LIN {X -0.060,Y -618.449,Z 1038.668,A 0.000,B 0.000,C 90.000,E1 336.230} C_DIS
LIN {X 0.200,Y -620.770,Z 1038.662,A 0.000,B 0.000,C 90.000,E1 335.177} C_DIS
LIN {X 0.196,Y -624.173,Z 1038.652,A 0.000,B 0.000,C 90.000,E1 333.384} C_DIS
LIN {X 0.244,Y -626.247,Z 1038.645,A 0.000,B 0.000,C 90.000,E1 332.103} C_DIS
LIN {X -0.253,Y -627.737,Z 1038.640,A 0.000,B 0.000,C 90.000,E1 331.129} C_DIS
LIN {X -0.406,Y -629.343,Z 1038.632,A 0.000,B 0.000,C 90.000,E1 329.871} C_DIS
LIN {X 0.333,Y -630.595,Z 1038.625,A 0.000,B 0.000,C 90.000,E1 328.535} C_DIS
LIN {X 0.027,Y -631.655,Z 1038.618,A 0.000,B 0.000,C 90.000,E1 327.296} C_DIS
LIN {X 0.271,Y -632.422,Z 1038.611,A 0.000,B 0.000,C 90.000,E1 326.008} C_DIS
LIN {X -0.015,Y -632.715,Z 1038.606,A 0.000,B 0.000,C 90.000,E1 325.022} C_DIS
LIN {X 0.076,Y -632.913,Z 1038.597,A 0.000,B 0.000,C 90.000,E1 323.497} C_DIS
LIN {X -0.098,Y -633.067,Z 1038.587,A 0.000,B 0.000,C 90.000,E1 321.743} C_DIS
LIN {X 0.257,Y -633.344,Z 1038.579,A 0.000,B 0.000,C 90.000,E1 320.194} C_DIS
LIN {X 0.129,Y -633.583,Z 1038.571,A 0.000,B 0.000,C 90.000,E1 318.690} C_DIS
LIN {X -0.259,Y -633.721,Z 1038.565,A 0.000,B 0.000,C 90.000,E1 317.715} C_DIS
LIN {X 0.356,Y -634.009,Z 1038.555,A 0.000,B 0.000,C 90.000,E1 315.891} C_DIS
LIN {X -0.368,Y -634.348,Z 1038.545,A 0.000,B 0.000,C 90.000,E1 314.190} C_DIS
LIN {X 0.114,Y -634.612,Z 1038.540,A 0.000,B 0.000,C 90.000,E1 313.137} C_DIS
LIN {X -0.371,Y -634.828,Z 1038.533,A 0.000,B 0.000,C 90.000,E1 311.919} C_DIS
LIN {X 0.051,Y -634.991,Z 1038.526,A 0.000,B 0.000,C 90.000,E1 310.620} C_DIS
LIN {X 0.204,Y -635.096,Z 1038.521,A 0.000,B 0.000,C 90.000,E1 309.850} C_DIS
LIN {X 0.329,Y -635.110,Z 1038.516,A 0.000,B 0.000,C 90.000,E1 308.830} C_DIS
LIN {X 0.074,Y -635.210,Z 1038.503,A 0.000,B 0.000,C 90.000,E1 306.583} C_DIS
LIN {X -0.174,Y -635.840,Z 1038.488,A 0.000,B 0.000,C 90.000,E1 303.833} C_DIS
LIN {X 0.041,Y -636.792,Z 1038.477,A 0.000,B 0.000,C 90.000,E1 301.799} C_DIS
LIN {X 0.088,Y -637.787,Z 1038.468,A 0.000,B 0.000,C 90.000,E1 300.285} C_DIS
LIN {X -0.030,Y -639.112,Z 1038.459,A 0.000,B 0.000,C 90.000,E1 298.537} C_DIS
LIN {X 0.261,Y -640.188,Z 1038.452,A 0.000,B 0.000,C 90.000,E1 297.257} C_DIS
LIN {X -0.061,Y -640.906,Z 1038.446,A 0.000,B 0.000,C 90.000,E1 296.283} C_DIS
LIN {X -0.147,Y -641.266,Z 1038.442,A 0.000,B 0.000,C 90.000,E1 295.540} C_DIS
LIN {X 0.117,Y -641.463,Z 1038.436,A 0.000,B 0.000,C 90.000,E1 294.515} C_DIS
LIN {X 0.111,Y -641.357,Z 1038.431,A 0.000,B 0.000,C 90.000,E1 293.515} C_DIS
LIN {X 0.102,Y -640.897,Z 1038.425,A 0.000,B 0.000,C 90.000,E1 292.514} C_DIS
LIN {X 0.029,Y -640.393,Z 1038.421,A 0.000,B 0.000,C 90.000,E1 291.770} C_DIS
LIN {X -0.154,Y -640.110,Z 1038.420,A 0.000,B 0.000,C 90.000,E1 291.535} C_DIS
LIN {X -0.284,Y -639.216,Z 1038.417,A 0.000,B 0.000,C 90.000,E1 291.046} C_DIS
LIN {X -0.192,Y -637.595,Z 1038.414,A 0.000,B 0.000,C 90.000,E1 290.536} C_DIS
LIN {X 0.222,Y -636.440,Z 1038.413,A 0.000,B 0.000,C 90.000,E1 290.248} C_DIS
LIN {X 0.069,Y -632.866,Z 1038.410,A 0.000,B 0.000,C 90.000,E1 289.758} C_DIS
LIN {X 0.078,Y -631.575,Z 1038.409,A 0.000,B 0.000,C 90.000,E1 289.631} C_DIS
LIN {X 0.157,Y -627.206,Z 1038.407,A 0.000,B 0.000,C 90.000,E1 289.268} C_DIS
LIN {X 0.365,Y -625.795,Z 1038.407,A 0.000,B 0.000,C 90.000,E1 289.141} C_DIS
LIN {X -0.222,Y -623.815,Z 1038.406,A 0.000,B 0.000,C 90.000,E1 289.087} C_DIS
LIN {X -0.131,Y -619.940,Z 1038.405,A 0.000,B 0.000,C 90.000,E1 288.906} C_DIS
LIN {X -0.205,Y -616.809,Z 1038.404,A 0.000,B 0.000,C 90.000,E1 288.725} C_DIS
LIN {X -0.172,Y -609.298,Z 1038.402,A 0.000,B 0.000,C 90.000,E1 288.417} C_DIS
LIN {X -0.167,Y -595.438,Z 1038.400,A 0.000,B 0.000,C 90.000,E1 287.928} C_DIS
LIN {X -0.153,Y -588.161,Z 1038.398,A 0.000,B 0.000,C 90.000,E1 287.692} C_DIS
LIN {X -0.073,Y -579.446,Z 1038.397,A 0.000,B 0.000,C 90.000,E1 287.402} C_DIS
LIN {X 0.070,Y -570.332,Z 1038.395,A 0.000,B 0.000,C 90.000,E1 287.040} C_DIS
LIN {X 0.055,Y -565.220,Z 1038.393,A 0.000,B 0.000,C 90.000,E1 286.804} C_DIS
LIN {X -0.217,Y -562.660,Z 1038.393,A 0.000,B 0.000,C 90.000,E1 286.677} C_DIS
LIN {X 0.099,Y -559.516,Z 1038.391,A 0.000,B 0.000,C 90.000,E1 286.441} C_DIS
LIN {X 0.192,Y -558.622,Z 1038.391,A 0.000,B 0.000,C 90.000,E1 286.315} C_DIS
LIN {X -0.205,Y -558.386,Z 1038.391,A 0.000,B 0.000,C 90.000,E1 286.315} C_DIS
LIN {X 0.290,Y -586.431,Z 1038.391,A 0.000,B 0.000,C 90.000,E1 286.260} C_DIS
LIN {X -0.354,Y -591.713,Z 1038.390,A 0.000,B 0.000,C 90.000,E1 286.205} C_DIS
LIN {X 0.109,Y -594.085,Z 1038.389,A 0.000,B 0.000,C 90.000,E1 286.079} C_DIS
LIN {X 0.215,Y -598.623,Z 1038.388,A 0.000,B 0.000,C 90.000,E1 285.733} C_DIS
LIN {X -0.132,Y -600.931,Z 1038.386,A 0.000,B 0.000,C 90.000,E1 285.552} C_DIS
LIN {X -0.291,Y -604.296,Z 1038.384,A 0.000,B 0.000,C 90.000,E1 285.190} C_DIS
LIN {X 0.020,Y -606.088,Z 1038.383,A 0.000,B 0.000,C 90.000,E1 284.898} C_DIS
LIN {X 0.233,Y -609.291,Z 1038.380,A 0.000,B 0.000,C 90.000,E1 284.356} C_DIS
LIN {X 0.115,Y -612.175,Z 1038.376,A 0.000,B 0.000,C 90.000,E1 283.716} C_DIS
LIN {X 0.359,Y -614.055,Z 1038.373,A 0.000,B 0.000,C 90.000,E1 283.175} C_DIS
LIN {X 0.115,Y -614.648,Z 1038.372,A 0.000,B 0.000,C 90.000,E1 282.939} C_DIS
LIN {X 0.233,Y -615.426,Z 1038.369,A 0.000,B 0.000,C 90.000,E1 282.411} C_DIS
LIN {X 0.230,Y -615.605,Z 1038.366,A 0.000,B 0.000,C 90.000,E1 281.895} C_DIS
LIN {X -0.244,Y -615.085,Z 1038.363,A 0.000,B 0.000,C 90.000,E1 281.422} C_DIS
LIN {X 0.121,Y -614.650,Z 1038.362,A 0.000,B 0.000,C 90.000,E1 281.130} C_DIS
LIN {X 0.242,Y -613.270,Z 1038.359,A 0.000,B 0.000,C 90.000,E1 280.602} C_DIS
LIN {X 0.240,Y -610.812,Z 1038.356,A 0.000,B 0.000,C 90.000,E1 280.084} C_DIS
LIN {X -0.269,Y -607.576,Z 1038.353,A 0.000,B 0.000,C 90.000,E1 279.613} C_DIS
LIN {X 0.065,Y -605.581,Z 1038.352,A 0.000,B 0.000,C 90.000,E1 279.321} C_DIS
LIN {X -0.142,Y -603.544,Z 1038.350,A 0.000,B 0.000,C 90.000,E1 279.095} C_DIS
LIN {X -0.232,Y -602.339,Z 1038.350,A 0.000,B 0.000,C 90.000,E1 278.973} C_DIS
LIN {X 0.150,Y -599.442,Z 1038.348,A 0.000,B 0.000,C 90.000,E1 278.690} C_DIS
LIN {X 0.085,Y -597.004,Z 1038.347,A 0.000,B 0.000,C 90.000,E1 278.454} C_DIS
LIN {X 0.092,Y -592.425,Z 1038.345,A 0.000,B 0.000,C 90.000,E1 278.106} C_DIS
LIN {X -0.161,Y -590.174,Z 1038.344,A 0.000,B 0.000,C 90.000,E1 277.936} C_DIS
LIN {X -0.137,Y -588.118,Z 1038.343,A 0.000,B 0.000,C 90.000,E1 277.814} C_DIS
LIN {X -0.193,Y -585.716,Z 1038.343,A 0.000,B 0.000,C 90.000,E1 277.701} C_DIS
LIN {X -0.111,Y -582.851,Z 1038.342,A 0.000,B 0.000,C 90.000,E1 277.530} C_DIS
LIN {X 0.253,Y -580.858,Z 1038.341,A 0.000,B 0.000,C 90.000,E1 277.409} C_DIS
LIN {X -0.022,Y -576.101,Z 1038.341,A 0.000,B 0.000,C 90.000,E1 277.296} C_DIS
LIN {X 0.270,Y -574.938,Z 1038.340,A 0.000,B 0.000,C 90.000,E1 277.239} C_DIS
LIN {X -0.235,Y -568.564,Z 1038.340,A 0.000,B 0.000,C 90.000,E1 277.239} C_DIS
LIN {X -0.270,Y -546.914,Z 1038.340,A 0.000,B 0.000,C 90.000,E1 277.239} C_DIS
LIN {X -0.073,Y -545.872,Z 1038.339,A 0.000,B 0.000,C 90.000,E1 277.068} C_DIS
LIN {X 0.058,Y -543.522,Z 1038.338,A 0.000,B 0.000,C 90.000,E1 276.777} C_DIS
LIN {X 0.016,Y -543.511,Z 1038.338,A 0.000,B 0.000,C 90.000,E1 276.777} C_DIS
LIN {X -0.061,Y -542.122,Z 1038.331,A 0.000,B 0.000,C 90.000,E1 275.511} C_DIS
LIN {X 0.194,Y -540.725,Z 1038.320,A 0.000,B 0.000,C 90.000,E1 273.498} C_DIS
LIN {X -0.170,Y -539.690,Z 1038.309,A 0.000,B 0.000,C 90.000,E1 271.547} C_DIS
LIN {X -0.101,Y -539.052,Z 1038.302,A 0.000,B 0.000,C 90.000,E1 270.401} C_DIS
LIN {X -0.026,Y -538.094,Z 1038.294,A 0.000,B 0.000,C 90.000,E1 268.969} C_DIS
LIN {X 0.054,Y -536.613,Z 1038.283,A 0.000,B 0.000,C 90.000,E1 266.963} C_DIS
LIN {X 0.125,Y -535.600,Z 1038.275,A 0.000,B 0.000,C 90.000,E1 265.527} C_DIS
LIN {X 0.220,Y -534.366,Z 1038.266,A 0.000,B 0.000,C 90.000,E1 263.799} C_DIS
LIN {X -0.264,Y -533.403,Z 1038.259,A 0.000,B 0.000,C 90.000,E1 262.704} C_DIS
LIN {X -0.121,Y -531.960,Z 1038.251,A 0.000,B 0.000,C 90.000,E1 261.254} C_DIS
LIN {X 0.109,Y -529.384,Z 1038.239,A 0.000,B 0.000,C 90.000,E1 258.926} C_DIS
LIN {X -0.212,Y -527.530,Z 1038.229,A 0.000,B 0.000,C 90.000,E1 257.229} C_DIS
LIN {X 0.050,Y -525.635,Z 1038.219,A 0.000,B 0.000,C 90.000,E1 255.463} C_DIS
LIN {X -0.116,Y -524.030,Z 1038.211,A 0.000,B 0.000,C 90.000,E1 254.031} C_DIS
LIN {X 0.192,Y -522.504,Z 1038.203,A 0.000,B 0.000,C 90.000,E1 252.543} C_DIS
LIN {X -0.026,Y -521.203,Z 1038.197,A 0.000,B 0.000,C 90.000,E1 251.402} C_DIS
LIN {X 0.018,Y -519.076,Z 1038.187,A 0.000,B 0.000,C 90.000,E1 249.645} C_DIS
LIN {X -0.096,Y -516.889,Z 1038.177,A 0.000,B 0.000,C 90.000,E1 247.901} C_DIS
LIN {X -0.232,Y -515.322,Z 1038.171,A 0.000,B 0.000,C 90.000,E1 246.741} C_DIS
LIN {X -0.113,Y -514.169,Z 1038.166,A 0.000,B 0.000,C 90.000,E1 245.845} C_DIS
LIN {X 0.015,Y -511.805,Z 1038.158,A 0.000,B 0.000,C 90.000,E1 244.357} C_DIS
LIN {X -0.025,Y -509.920,Z 1038.151,A 0.000,B 0.000,C 90.000,E1 243.179} C_DIS
LIN {X 0.133,Y -507.929,Z 1038.144,A 0.000,B 0.000,C 90.000,E1 241.975} C_DIS
LIN {X -0.077,Y -505.267,Z 1038.136,A 0.000,B 0.000,C 90.000,E1 240.511} C_DIS
LIN {X 0.110,Y -502.587,Z 1038.128,A 0.000,B 0.000,C 90.000,E1 238.997} C_DIS
LIN {X 0.096,Y -499.218,Z 1038.118,A 0.000,B 0.000,C 90.000,E1 237.199} C_DIS
LIN {X -0.015,Y -496.865,Z 1038.111,A 0.000,B 0.000,C 90.000,E1 236.008} C_DIS
LIN {X -0.034,Y -492.964,Z 1038.101,A 0.000,B 0.000,C 90.000,E1 234.196} C_DIS
LIN {X -0.092,Y -489.440,Z 1038.093,A 0.000,B 0.000,C 90.000,E1 232.683} C_DIS
LIN {X -0.056,Y -483.684,Z 1038.079,A 0.000,B 0.000,C 90.000,E1 230.231} C_DIS
LIN {X -0.125,Y -478.929,Z 1038.067,A 0.000,B 0.000,C 90.000,E1 228.081} C_DIS
LIN {X -0.202,Y -475.740,Z 1038.058,A 0.000,B 0.000,C 90.000,E1 226.539} C_DIS
LIN {X -0.166,Y -471.201,Z 1038.046,A 0.000,B 0.000,C 90.000,E1 224.352} C_DIS
LIN {X 0.081,Y -466.692,Z 1038.034,A 0.000,B 0.000,C 90.000,E1 222.123} C_DIS
LIN {X 0.122,Y -463.522,Z 1038.025,A 0.000,B 0.000,C 90.000,E1 220.539} C_DIS
LIN {X -0.158,Y -459.461,Z 1038.015,A 0.000,B 0.000,C 90.000,E1 218.669} C_DIS
LIN {X -0.187,Y -455.999,Z 1038.006,A 0.000,B 0.000,C 90.000,E1 217.076} C_DIS
LIN {X 0.077,Y -452.503,Z 1037.997,A 0.000,B 0.000,C 90.000,E1 215.438} C_DIS
LIN {X -0.035,Y -450.542,Z 1037.992,A 0.000,B 0.000,C 90.000,E1 214.485} C_DIS
LIN {X -0.066,Y -446.481,Z 1037.981,A 0.000,B 0.000,C 90.000,E1 212.546} C_DIS
LIN {X -0.065,Y -442.186,Z 1037.970,A 0.000,B 0.000,C 90.000,E1 210.590} C_DIS
LIN {X -0.089,Y -439.234,Z 1037.963,A 0.000,B 0.000,C 90.000,E1 209.283} C_DIS
LIN {X -0.155,Y -436.188,Z 1037.955,A 0.000,B 0.000,C 90.000,E1 207.975} C_DIS
LIN {X -0.063,Y -431.773,Z 1037.944,A 0.000,B 0.000,C 90.000,E1 205.976} C_DIS
LIN {X 0.113,Y -426.007,Z 1037.929,A 0.000,B 0.000,C 90.000,E1 203.281} C_DIS
LIN {X -0.057,Y -420.811,Z 1037.915,A 0.000,B 0.000,C 90.000,E1 200.610} C_DIS
LIN {X -0.196,Y -413.886,Z 1037.890,A 0.000,B 0.000,C 90.000,E1 196.205} C_DIS
LIN {X -0.121,Y -411.969,Z 1037.880,A 0.000,B 0.000,C 90.000,E1 194.481} C_DIS
LIN {X 0.161,Y -411.252,Z 1037.875,A 0.000,B 0.000,C 90.000,E1 193.411} C_DIS
LIN {X -0.066,Y -410.760,Z 1037.869,A 0.000,B 0.000,C 90.000,E1 192.411} C_DIS
LIN {X -0.010,Y -411.012,Z 1037.865,A 0.000,B 0.000,C 90.000,E1 191.715} C_DIS
LIN {X 0.020,Y -411.285,Z 1037.863,A 0.000,B 0.000,C 90.000,E1 191.366} C_DIS
LIN {X 0.130,Y -411.738,Z 1037.861,A 0.000,B 0.000,C 90.000,E1 191.007} C_DIS
LIN {X -0.141,Y -413.356,Z 1037.858,A 0.000,B 0.000,C 90.000,E1 190.366} C_DIS
LIN {X -0.105,Y -414.633,Z 1037.856,A 0.000,B 0.000,C 90.000,E1 190.018} C_DIS
LIN {X -0.071,Y -416.767,Z 1037.853,A 0.000,B 0.000,C 90.000,E1 189.500} C_DIS
LIN {X -0.076,Y -419.086,Z 1037.850,A 0.000,B 0.000,C 90.000,E1 189.095} C_DIS
LIN {X 0.050,Y -422.248,Z 1037.848,A 0.000,B 0.000,C 90.000,E1 188.568} C_DIS
LIN {X -0.094,Y -435.430,Z 1037.838,A 0.000,B 0.000,C 90.000,E1 186.777} C_DIS
LIN {X -0.176,Y -442.951,Z 1037.832,A 0.000,B 0.000,C 90.000,E1 185.796} C_DIS
LIN {X 0.050,Y -453.968,Z 1037.824,A 0.000,B 0.000,C 90.000,E1 184.302} C_DIS
LIN {X -0.211,Y -462.264,Z 1037.818,A 0.000,B 0.000,C 90.000,E1 183.212} C_DIS
LIN {X -0.110,Y -472.302,Z 1037.810,A 0.000,B 0.000,C 90.000,E1 181.776} C_DIS
LIN {X 0.235,Y -481.700,Z 1037.802,A 0.000,B 0.000,C 90.000,E1 180.344} C_DIS
LIN {X 0.172,Y -487.705,Z 1037.797,A 0.000,B 0.000,C 90.000,E1 179.427} C_DIS
LIN {X -0.149,Y -494.571,Z 1037.791,A 0.000,B 0.000,C 90.000,E1 178.396} C_DIS
LIN {X -0.056,Y -500.306,Z 1037.786,A 0.000,B 0.000,C 90.000,E1 177.478} C_DIS
LIN {X 0.111,Y -507.412,Z 1037.779,A 0.000,B 0.000,C 90.000,E1 176.274} C_DIS
LIN {X 0.222,Y -516.017,Z 1037.771,A 0.000,B 0.000,C 90.000,E1 174.780} C_DIS
LIN {X 0.026,Y -524.489,Z 1037.763,A 0.000,B 0.000,C 90.000,E1 173.337} C_DIS
LIN {X -0.017,Y -532.743,Z 1037.755,A 0.000,B 0.000,C 90.000,E1 171.894} C_DIS
LIN {X -0.112,Y -541.531,Z 1037.746,A 0.000,B 0.000,C 90.000,E1 170.330} C_DIS
LIN {X 0.057,Y -550.142,Z 1037.738,A 0.000,B 0.000,C 90.000,E1 168.757} C_DIS
LIN {X -0.007,Y -558.485,Z 1037.729,A 0.000,B 0.000,C 90.000,E1 167.229} C_DIS
LIN {X 0.299,Y -563.558,Z 1037.724,A 0.000,B 0.000,C 90.000,E1 166.228} C_DIS
LIN {X 0.181,Y -570.648,Z 1037.716,A 0.000,B 0.000,C 90.000,E1 164.866} C_DIS
LIN {X 0.081,Y -575.369,Z 1037.711,A 0.000,B 0.000,C 90.000,E1 163.921} C_DIS
LIN {X 0.198,Y -579.985,Z 1037.705,A 0.000,B 0.000,C 90.000,E1 162.960} C_DIS
LIN {X -0.184,Y -584.304,Z 1037.700,A 0.000,B 0.000,C 90.000,E1 162.054} C_DIS
LIN {X -0.032,Y -588.964,Z 1037.694,A 0.000,B 0.000,C 90.000,E1 160.967} C_DIS
LIN {X 0.066,Y -594.393,Z 1037.687,A 0.000,B 0.000,C 90.000,E1 159.625} C_DIS
LIN {X -0.211,Y -598.419,Z 1037.681,A 0.000,B 0.000,C 90.000,E1 158.592} C_DIS
LIN {X 0.262,Y -603.058,Z 1037.674,A 0.000,B 0.000,C 90.000,E1 157.230} C_DIS
LIN {X -0.238,Y -606.530,Z 1037.668,A 0.000,B 0.000,C 90.000,E1 156.230} C_DIS
LIN {X -0.143,Y -609.792,Z 1037.662,A 0.000,B 0.000,C 90.000,E1 155.177} C_DIS
LIN {X -0.305,Y -612.814,Z 1037.656,A 0.000,B 0.000,C 90.000,E1 154.152} C_DIS
LIN {X 0.104,Y -616.332,Z 1037.649,A 0.000,B 0.000,C 90.000,E1 152.820} C_DIS
LIN {X 0.319,Y -619.009,Z 1037.643,A 0.000,B 0.000,C 90.000,E1 151.769} C_DIS
LIN {X 0.031,Y -622.879,Z 1037.635,A 0.000,B 0.000,C 90.000,E1 150.255} C_DIS
LIN {X -0.190,Y -626.033,Z 1037.628,A 0.000,B 0.000,C 90.000,E1 148.997} C_DIS
LIN {X -0.034,Y -629.093,Z 1037.621,A 0.000,B 0.000,C 90.000,E1 147.709} C_DIS
LIN {X 0.185,Y -632.629,Z 1037.612,A 0.000,B 0.000,C 90.000,E1 146.167} C_DIS
LIN {X -0.231,Y -636.111,Z 1037.604,A 0.000,B 0.000,C 90.000,E1 144.689} C_DIS
LIN {X 0.317,Y -639.575,Z 1037.595,A 0.000,B 0.000,C 90.000,E1 143.130} C_DIS
LIN {X -0.081,Y -643.088,Z 1037.587,A 0.000,B 0.000,C 90.000,E1 141.662} C_DIS
LIN {X 0.010,Y -647.078,Z 1037.577,A 0.000,B 0.000,C 90.000,E1 139.908} C_DIS
LIN {X 0.108,Y -651.094,Z 1037.568,A 0.000,B 0.000,C 90.000,E1 138.162} C_DIS
LIN {X -0.268,Y -656.433,Z 1037.555,A 0.000,B 0.000,C 90.000,E1 135.972} C_DIS
LIN {X -0.054,Y -663.721,Z 1037.540,A 0.000,B 0.000,C 90.000,E1 133.257} C_DIS
LIN {X -0.098,Y -667.183,Z 1037.534,A 0.000,B 0.000,C 90.000,E1 132.043} C_DIS
LIN {X -0.048,Y -670.668,Z 1037.527,A 0.000,B 0.000,C 90.000,E1 130.825} C_DIS
LIN {X 0.156,Y -674.730,Z 1037.519,A 0.000,B 0.000,C 90.000,E1 129.358} C_DIS
LIN {X -0.097,Y -678.022,Z 1037.512,A 0.000,B 0.000,C 90.000,E1 128.177} C_DIS
LIN {X -0.139,Y -682.350,Z 1037.503,A 0.000,B 0.000,C 90.000,E1 126.503} C_DIS
LIN {X 0.432,Y -686.073,Z 1037.495,A 0.000,B 0.000,C 90.000,E1 125.025} C_DIS
LIN {X 0.116,Y -689.677,Z 1037.487,A 0.000,B 0.000,C 90.000,E1 123.627} C_DIS
LIN {X 0.065,Y -693.179,Z 1037.479,A 0.000,B 0.000,C 90.000,E1 122.212} C_DIS
LIN {X 0.192,Y -695.373,Z 1037.474,A 0.000,B 0.000,C 90.000,E1 121.258} C_DIS
LIN {X 0.241,Y -697.851,Z 1037.467,A 0.000,B 0.000,C 90.000,E1 120.079} C_DIS
LIN {X -0.193,Y -699.002,Z 1037.463,A 0.000,B 0.000,C 90.000,E1 119.411} C_DIS
LIN {X -0.085,Y -700.557,Z 1037.457,A 0.000,B 0.000,C 90.000,E1 118.231} C_DIS
LIN {X -0.350,Y -702.425,Z 1037.448,A 0.000,B 0.000,C 90.000,E1 116.616} C_DIS
LIN {X 0.116,Y -703.430,Z 1037.441,A 0.000,B 0.000,C 90.000,E1 115.412} C_DIS
LIN {X 0.031,Y -703.903,Z 1037.437,A 0.000,B 0.000,C 90.000,E1 114.719} C_DIS
LIN {X -0.044,Y -703.825,Z 1037.435,A 0.000,B 0.000,C 90.000,E1 114.259} C_DIS
LIN {X -0.049,Y -703.663,Z 1037.433,A 0.000,B 0.000,C 90.000,E1 114.027} C_DIS
LIN {X -0.131,Y -702.667,Z 1037.431,A 0.000,B 0.000,C 90.000,E1 113.567} C_DIS
LIN {X -0.134,Y -701.822,Z 1037.430,A 0.000,B 0.000,C 90.000,E1 113.334} C_DIS
LIN {X 0.138,Y -699.031,Z 1037.427,A 0.000,B 0.000,C 90.000,E1 112.845} C_DIS
LIN {X -0.374,Y -698.143,Z 1037.426,A 0.000,B 0.000,C 90.000,E1 112.770} C_DIS
LIN {X -0.242,Y -696.824,Z 1037.426,A 0.000,B 0.000,C 90.000,E1 112.642} C_DIS
LIN {X 0.161,Y -692.932,Z 1037.424,A 0.000,B 0.000,C 90.000,E1 112.386} C_DIS
LIN {X 0.326,Y -689.873,Z 1037.424,A 0.000,B 0.000,C 90.000,E1 112.206} C_DIS
LIN {X -0.046,Y -688.040,Z 1037.423,A 0.000,B 0.000,C 90.000,E1 112.153} C_DIS
LIN {X -0.156,Y -685.469,Z 1037.423,A 0.000,B 0.000,C 90.000,E1 112.078} C_DIS
LIN {X -0.191,Y -682.766,Z 1037.422,A 0.000,B 0.000,C 90.000,E1 112.025} C_DIS
LIN {X 0.323,Y -675.461,Z 1037.422,A 0.000,B 0.000,C 90.000,E1 111.897} C_DIS
LIN {X 0.249,Y -611.830,Z 1037.422,A 0.000,B 0.000,C 90.000,E1 111.897} C_DIS
LIN {X -0.103,Y -603.967,Z 1037.420,A 0.000,B 0.000,C 90.000,E1 111.663} C_DIS
LIN {X -0.084,Y -597.881,Z 1037.419,A 0.000,B 0.000,C 90.000,E1 111.354} C_DIS
LIN {X 0.117,Y -592.278,Z 1037.417,A 0.000,B 0.000,C 90.000,E1 110.972} C_DIS
LIN {X 0.178,Y -585.389,Z 1037.414,A 0.000,B 0.000,C 90.000,E1 110.429} C_DIS
LIN {X -0.147,Y -577.122,Z 1037.410,A 0.000,B 0.000,C 90.000,E1 109.758} C_DIS
LIN {X 0.193,Y -571.004,Z 1037.407,A 0.000,B 0.000,C 90.000,E1 109.268} C_DIS
LIN {X -0.352,Y -569.434,Z 1037.407,A 0.000,B 0.000,C 90.000,E1 109.214} C_DIS
LIN {X -0.255,Y -561.218,Z 1037.404,A 0.000,B 0.000,C 90.000,E1 108.725} C_DIS
LIN {X -0.158,Y -554.609,Z 1037.402,A 0.000,B 0.000,C 90.000,E1 108.362} C_DIS
LIN {X 0.138,Y -549.479,Z 1037.400,A 0.000,B 0.000,C 90.000,E1 108.000} C_DIS
LIN {X 0.108,Y -548.012,Z 1037.399,A 0.000,B 0.000,C 90.000,E1 107.819} C_DIS
LIN {X 0.067,Y -547.994,Z 1037.399,A 0.000,B 0.000,C 90.000,E1 107.819} C_DIS
LIN {X -0.157,Y -547.523,Z 1037.398,A 0.000,B 0.000,C 90.000,E1 107.583} C_DIS
LIN {X -0.026,Y -547.592,Z 1037.394,A 0.000,B 0.000,C 90.000,E1 106.985} C_DIS
LIN {X 0.031,Y -548.185,Z 1037.390,A 0.000,B 0.000,C 90.000,E1 106.134} C_DIS
LIN {X 0.044,Y -549.401,Z 1037.377,A 0.000,B 0.000,C 90.000,E1 103.883} C_DIS
LIN {X -0.230,Y -552.195,Z 1037.359,A 0.000,B 0.000,C 90.000,E1 100.546} C_DIS
LIN {X 0.138,Y -554.945,Z 1037.344,A 0.000,B 0.000,C 90.000,E1 97.992} C_DIS
LIN {X 0.068,Y -556.523,Z 1037.337,A 0.000,B 0.000,C 90.000,E1 96.606} C_DIS
LIN {X 0.020,Y -557.995,Z 1037.329,A 0.000,B 0.000,C 90.000,E1 95.220} C_DIS
LIN {X -0.182,Y -558.849,Z 1037.323,A 0.000,B 0.000,C 90.000,E1 94.131} C_DIS
LIN {X 0.107,Y -559.464,Z 1037.318,A 0.000,B 0.000,C 90.000,E1 93.269} C_DIS
LIN {X 0.131,Y -560.249,Z 1037.309,A 0.000,B 0.000,C 90.000,E1 91.604} C_DIS
LIN {X 0.134,Y -560.857,Z 1037.300,A 0.000,B 0.000,C 90.000,E1 89.943} C_DIS
LIN {X 0.264,Y -561.537,Z 1037.289,A 0.000,B 0.000,C 90.000,E1 87.993} C_DIS
LIN {X 0.213,Y -561.973,Z 1037.281,A 0.000,B 0.000,C 90.000,E1 86.617} C_DIS
LIN {X -0.261,Y -562.515,Z 1037.272,A 0.000,B 0.000,C 90.000,E1 85.008} C_DIS
LIN {X -0.265,Y -562.849,Z 1037.265,A 0.000,B 0.000,C 90.000,E1 83.628} C_DIS
LIN {X -0.218,Y -563.471,Z 1037.251,A 0.000,B 0.000,C 90.000,E1 81.141} C_DIS
LIN {X 0.041,Y -564.402,Z 1037.237,A 0.000,B 0.000,C 90.000,E1 78.634} C_DIS
LIN {X -0.112,Y -565.670,Z 1037.223,A 0.000,B 0.000,C 90.000,E1 76.172} C_DIS
LIN {X 0.251,Y -566.946,Z 1037.213,A 0.000,B 0.000,C 90.000,E1 74.212} C_DIS
LIN {X -0.067,Y -568.242,Z 1037.203,A 0.000,B 0.000,C 90.000,E1 72.598} C_DIS
LIN {X -0.150,Y -569.133,Z 1037.197,A 0.000,B 0.000,C 90.000,E1 71.511} C_DIS
LIN {X 0.127,Y -570.222,Z 1037.190,A 0.000,B 0.000,C 90.000,E1 70.115} C_DIS
LIN {X 0.062,Y -570.981,Z 1037.184,A 0.000,B 0.000,C 90.000,E1 69.028} C_DIS
LIN {X 0.031,Y -571.988,Z 1037.176,A 0.000,B 0.000,C 90.000,E1 67.667} C_DIS
LIN {X -0.150,Y -572.968,Z 1037.167,A 0.000,B 0.000,C 90.000,E1 66.049} C_DIS
LIN {X -0.239,Y -573.995,Z 1037.156,A 0.000,B 0.000,C 90.000,E1 64.152} C_DIS
LIN {X 0.259,Y -574.647,Z 1037.149,A 0.000,B 0.000,C 90.000,E1 62.743} C_DIS
LIN {X 0.254,Y -575.221,Z 1037.141,A 0.000,B 0.000,C 90.000,E1 61.385} C_DIS
LIN {X -0.275,Y -575.983,Z 1037.131,A 0.000,B 0.000,C 90.000,E1 59.537} C_DIS
LIN {X 0.176,Y -576.371,Z 1037.125,A 0.000,B 0.000,C 90.000,E1 58.408} C_DIS
LIN {X 0.287,Y -576.819,Z 1037.117,A 0.000,B 0.000,C 90.000,E1 57.041} C_DIS
LIN {X -0.070,Y -577.162,Z 1037.110,A 0.000,B 0.000,C 90.000,E1 55.722} C_DIS
LIN {X 0.068,Y -577.322,Z 1037.105,A 0.000,B 0.000,C 90.000,E1 54.895} C_DIS
LIN {X 0.054,Y -577.397,Z 1037.098,A 0.000,B 0.000,C 90.000,E1 53.543} C_DIS
LIN {X -0.277,Y -577.371,Z 1037.093,A 0.000,B 0.000,C 90.000,E1 52.763} C_DIS
LIN {X 0.039,Y -577.329,Z 1037.090,A 0.000,B 0.000,C 90.000,E1 52.190} C_DIS
LIN {X 0.058,Y -577.136,Z 1037.085,A 0.000,B 0.000,C 90.000,E1 51.376} C_DIS
LIN {X 0.093,Y -576.333,Z 1037.076,A 0.000,B 0.000,C 90.000,E1 49.747} C_DIS
LIN {X -0.188,Y -575.728,Z 1037.070,A 0.000,B 0.000,C 90.000,E1 48.690} C_DIS
LIN {X 0.192,Y -575.139,Z 1037.066,A 0.000,B 0.000,C 90.000,E1 47.838} C_DIS
LIN {X -0.010,Y -573.994,Z 1037.058,A 0.000,B 0.000,C 90.000,E1 46.500} C_DIS
LIN {X 0.348,Y -573.110,Z 1037.054,A 0.000,B 0.000,C 90.000,E1 45.648} C_DIS
LIN {X -0.306,Y -571.152,Z 1037.046,A 0.000,B 0.000,C 90.000,E1 44.352} C_DIS
LIN {X 0.110,Y -569.327,Z 1037.040,A 0.000,B 0.000,C 90.000,E1 43.218} C_DIS
LIN {X 0.105,Y -567.253,Z 1037.034,A 0.000,B 0.000,C 90.000,E1 42.123} C_DIS
LIN {X 0.009,Y -565.428,Z 1037.030,A 0.000,B 0.000,C 90.000,E1 41.310} C_DIS
LIN {X -0.056,Y -562.596,Z 1037.023,A 0.000,B 0.000,C 90.000,E1 40.216} C_DIS
LIN {X 0.141,Y -561.053,Z 1037.020,A 0.000,B 0.000,C 90.000,E1 39.644} C_DIS
LIN {X -0.009,Y -558.443,Z 1037.016,A 0.000,B 0.000,C 90.000,E1 38.830} C_DIS
LIN {X -0.187,Y -555.641,Z 1037.011,A 0.000,B 0.000,C 90.000,E1 38.016} C_DIS
LIN {X 0.042,Y -552.379,Z 1037.006,A 0.000,B 0.000,C 90.000,E1 37.156} C_DIS
LIN {X 0.234,Y -548.863,Z 1037.002,A 0.000,B 0.000,C 90.000,E1 36.297} C_DIS
LIN {X 0.066,Y -545.045,Z 1036.997,A 0.000,B 0.000,C 90.000,E1 35.471} C_DIS
LIN {X 0.169,Y -540.820,Z 1036.992,A 0.000,B 0.000,C 90.000,E1 34.612} C_DIS
LIN {X 0.061,Y -537.073,Z 1036.989,A 0.000,B 0.000,C 90.000,E1 33.913} C_DIS
LIN {X 0.068,Y -531.545,Z 1036.983,A 0.000,B 0.000,C 90.000,E1 32.911} C_DIS
LIN {X 0.031,Y -528.155,Z 1036.980,A 0.000,B 0.000,C 90.000,E1 32.339} C_DIS
LIN {X 0.250,Y -523.645,Z 1036.976,A 0.000,B 0.000,C 90.000,E1 31.592} C_DIS
LIN {X 0.155,Y -518.831,Z 1036.972,A 0.000,B 0.000,C 90.000,E1 30.875} C_DIS
LIN {X -0.251,Y -514.730,Z 1036.968,A 0.000,B 0.000,C 90.000,E1 30.335} C_DIS
LIN {X 0.279,Y -509.188,Z 1036.964,A 0.000,B 0.000,C 90.000,E1 29.539} C_DIS
LIN {X 0.245,Y -504.407,Z 1036.961,A 0.000,B 0.000,C 90.000,E1 28.949} C_DIS
LIN {X -0.144,Y -496.495,Z 1036.956,A 0.000,B 0.000,C 90.000,E1 28.103} C_DIS
LIN {X 0.172,Y -489.642,Z 1036.952,A 0.000,B 0.000,C 90.000,E1 27.334} C_DIS
LIN {X 0.131,Y -479.801,Z 1036.947,A 0.000,B 0.000,C 90.000,E1 26.360} C_DIS
LIN {X 0.173,Y -469.817,Z 1036.941,A 0.000,B 0.000,C 90.000,E1 25.412} C_DIS
LIN {X -0.155,Y -462.233,Z 1036.938,A 0.000,B 0.000,C 90.000,E1 24.771} C_DIS
LIN {X 0.239,Y -454.776,Z 1036.934,A 0.000,B 0.000,C 90.000,E1 24.079} C_DIS
LIN {X -0.148,Y -429.296,Z 1036.922,A 0.000,B 0.000,C 90.000,E1 21.897} C_DIS
LIN {X -0.083,Y -416.288,Z 1036.914,A 0.000,B 0.000,C 90.000,E1 20.610} C_DIS
LIN {X 0.084,Y -403.873,Z 1036.907,A 0.000,B 0.000,C 90.000,E1 19.214} C_DIS
LIN {X 0.163,Y -399.929,Z 1036.904,A 0.000,B 0.000,C 90.000,E1 18.725} C_DIS
LIN {X 0.068,Y -395.635,Z 1036.901,A 0.000,B 0.000,C 90.000,E1 18.127} C_DIS
LIN {X 0.024,Y -393.301,Z 1036.898,A 0.000,B 0.000,C 90.000,E1 17.692} C_DIS
LIN {X 0.128,Y -391.875,Z 1036.896,A 0.000,B 0.000,C 90.000,E1 17.166} C_DIS
LIN {X 0.139,Y -391.439,Z 1036.894,A 0.000,B 0.000,C 90.000,E1 16.804} C_DIS
LIN {X 0.163,Y -391.286,Z 1036.893,A 0.000,B 0.000,C 90.000,E1 16.622} C_DIS
LIN {X -0.152,Y -391.430,Z 1036.888,A 0.000,B 0.000,C 90.000,E1 15.898} C_DIS
LIN {X 0.189,Y -396.870,Z 1036.863,A 0.000,B 0.000,C 90.000,E1 11.243} C_DIS
LIN {X -0.056,Y -403.950,Z 1036.839,A 0.000,B 0.000,C 90.000,E1 7.068} C_DIS
LIN {X -0.113,Y -409.067,Z 1036.826,A 0.000,B 0.000,C 90.000,E1 4.645} C_DIS
LIN {X -0.144,Y -412.059,Z 1036.818,A 0.000,B 0.000,C 90.000,E1 3.269} C_DIS
LIN {X -0.128,Y -414.356,Z 1036.814,A 0.000,B 0.000,C 90.000,E1 2.579} C_DIS
LIN {X -0.066,Y -417.745,Z 1036.811,A 0.000,B 0.000,C 90.000,E1 1.949} C_DIS
LIN {X -0.120,Y -421.520,Z 1036.809,A 0.000,B 0.000,C 90.000,E1 1.547} C_DIS
LIN {X 0.012,Y -423.260,Z 1036.808,A 0.000,B 0.000,C 90.000,E1 1.375} C_DIS
LIN {X -0.175,Y -428.885,Z 1036.806,A 0.000,B 0.000,C 90.000,E1 1.031} C_DIS
LIN {X 0.177,Y -438.428,Z 1036.802,A 0.000,B 0.000,C 90.000,E1 0.401} C_DIS
LIN {X 0.123,Y -461.820,Z 1036.794,A 0.000,B 0.000,C 90.000,E1 358.969} C_DIS
LIN {X 0.095,Y -473.331,Z 1036.791,A 0.000,B 0.000,C 90.000,E1 358.282} C_DIS
LIN {X -0.089,Y -489.758,Z 1036.785,A 0.000,B 0.000,C 90.000,E1 357.306} C_DIS
LIN {X -0.203,Y -500.945,Z 1036.781,A 0.000,B 0.000,C 90.000,E1 356.617} C_DIS
LIN {X 0.192,Y -507.176,Z 1036.779,A 0.000,B 0.000,C 90.000,E1 356.159} C_DIS
LIN {X -0.020,Y -514.934,Z 1036.776,A 0.000,B 0.000,C 90.000,E1 355.641} C_DIS
LIN {X 0.022,Y -523.809,Z 1036.772,A 0.000,B 0.000,C 90.000,E1 354.951} C_DIS
LIN {X -0.225,Y -531.007,Z 1036.769,A 0.000,B 0.000,C 90.000,E1 354.375} C_DIS
LIN {X -0.248,Y -537.785,Z 1036.765,A 0.000,B 0.000,C 90.000,E1 353.742} C_DIS
LIN {X 0.174,Y -543.099,Z 1036.762,A 0.000,B 0.000,C 90.000,E1 353.166} C_DIS
LIN {X 0.245,Y -549.349,Z 1036.758,A 0.000,B 0.000,C 90.000,E1 352.470} C_DIS
LIN {X 0.125,Y -554.927,Z 1036.755,A 0.000,B 0.000,C 90.000,E1 351.781} C_DIS
LIN {X -0.173,Y -559.024,Z 1036.751,A 0.000,B 0.000,C 90.000,E1 351.254} C_DIS
LIN {X -0.132,Y -563.618,Z 1036.748,A 0.000,B 0.000,C 90.000,E1 350.557} C_DIS
LIN {X -0.048,Y -567.765,Z 1036.744,A 0.000,B 0.000,C 90.000,E1 349.859} C_DIS
LIN {X 0.072,Y -571.628,Z 1036.740,A 0.000,B 0.000,C 90.000,E1 349.162} C_DIS
LIN {X 0.101,Y -575.969,Z 1036.735,A 0.000,B 0.000,C 90.000,E1 348.342} C_DIS
LIN {X 0.178,Y -579.845,Z 1036.731,A 0.000,B 0.000,C 90.000,E1 347.521} C_DIS
LIN {X -0.042,Y -584.576,Z 1036.725,A 0.000,B 0.000,C 90.000,E1 346.464} C_DIS
LIN {X -0.211,Y -589.043,Z 1036.719,A 0.000,B 0.000,C 90.000,E1 345.408} C_DIS
LIN {X 0.135,Y -592.285,Z 1036.714,A 0.000,B 0.000,C 90.000,E1 344.574} C_DIS
LIN {X 0.220,Y -596.432,Z 1036.708,A 0.000,B 0.000,C 90.000,E1 343.504} C_DIS
LIN {X 0.076,Y -599.434,Z 1036.704,A 0.000,B 0.000,C 90.000,E1 342.725} C_DIS
LIN {X -0.135,Y -603.201,Z 1036.698,A 0.000,B 0.000,C 90.000,E1 341.692} C_DIS
LIN {X 0.283,Y -606.699,Z 1036.693,A 0.000,B 0.000,C 90.000,E1 340.604} C_DIS
LIN {X 0.174,Y -609.914,Z 1036.687,A 0.000,B 0.000,C 90.000,E1 339.571} C_DIS
LIN {X 0.059,Y -613.578,Z 1036.679,A 0.000,B 0.000,C 90.000,E1 338.284} C_DIS
LIN {X -0.279,Y -615.658,Z 1036.675,A 0.000,B 0.000,C 90.000,E1 337.539} C_DIS
LIN {X -0.051,Y -618.194,Z 1036.669,A 0.000,B 0.000,C 90.000,E1 336.485} C_DIS
LIN {X -0.360,Y -620.563,Z 1036.664,A 0.000,B 0.000,C 90.000,E1 335.485} C_DIS
LIN {X 0.187,Y -622.150,Z 1036.659,A 0.000,B 0.000,C 90.000,E1 334.665} C_DIS
LIN {X 0.202,Y -624.587,Z 1036.652,A 0.000,B 0.000,C 90.000,E1 333.384} C_DIS
LIN {X 0.243,Y -626.327,Z 1036.647,A 0.000,B 0.000,C 90.000,E1 332.359} C_DIS
LIN {X -0.234,Y -628.212,Z 1036.640,A 0.000,B 0.000,C 90.000,E1 331.129} C_DIS
LIN {X -0.379,Y -629.832,Z 1036.632,A 0.000,B 0.000,C 90.000,E1 329.871} C_DIS
LIN {X -0.170,Y -631.155,Z 1036.625,A 0.000,B 0.000,C 90.000,E1 328.584} C_DIS
LIN {X -0.270,Y -632.236,Z 1036.618,A 0.000,B 0.000,C 90.000,E1 327.327} C_DIS
LIN {X 0.327,Y -633.062,Z 1036.611,A 0.000,B 0.000,C 90.000,E1 326.008} C_DIS
LIN {X 0.049,Y -633.445,Z 1036.606,A 0.000,B 0.000,C 90.000,E1 325.022} C_DIS
LIN {X 0.156,Y -633.686,Z 1036.597,A 0.000,B 0.000,C 90.000,E1 323.497} C_DIS
LIN {X 0.122,Y -633.848,Z 1036.589,A 0.000,B 0.000,C 90.000,E1 321.984} C_DIS
LIN {X -0.034,Y -634.185,Z 1036.579,A 0.000,B 0.000,C 90.000,E1 320.231} C_DIS
LIN {X 0.260,Y -634.471,Z 1036.571,A 0.000,B 0.000,C 90.000,E1 318.690} C_DIS
LIN {X -0.117,Y -634.643,Z 1036.565,A 0.000,B 0.000,C 90.000,E1 317.715} C_DIS
LIN {X -0.377,Y -634.993,Z 1036.555,A 0.000,B 0.000,C 90.000,E1 315.972} C_DIS
LIN {X -0.181,Y -635.390,Z 1036.545,A 0.000,B 0.000,C 90.000,E1 314.190} C_DIS
LIN {X -0.020,Y -635.677,Z 1036.541,A 0.000,B 0.000,C 90.000,E1 313.419} C_DIS
LIN {X -0.151,Y -635.976,Z 1036.533,A 0.000,B 0.000,C 90.000,E1 311.919} C_DIS
LIN {X -0.333,Y -636.313,Z 1036.523,A 0.000,B 0.000,C 90.000,E1 310.172} C_DIS
LIN {X 0.213,Y -636.365,Z 1036.517,A 0.000,B 0.000,C 90.000,E1 309.116} C_DIS
LIN {X 0.380,Y -636.515,Z 1036.504,A 0.000,B 0.000,C 90.000,E1 306.583} C_DIS
LIN {X 0.178,Y -637.147,Z 1036.488,A 0.000,B 0.000,C 90.000,E1 303.833} C_DIS
LIN {X -0.070,Y -638.271,Z 1036.476,A 0.000,B 0.000,C 90.000,E1 301.592} C_DIS
LIN {X 0.006,Y -639.323,Z 1036.467,A 0.000,B 0.000,C 90.000,E1 300.079} C_DIS
LIN {X 0.175,Y -640.715,Z 1036.457,A 0.000,B 0.000,C 90.000,E1 298.309} C_DIS
LIN {X -0.063,Y -641.846,Z 1036.450,A 0.000,B 0.000,C 90.000,E1 297.078} C_DIS
LIN {X 0.218,Y -642.537,Z 1036.445,A 0.000,B 0.000,C 90.000,E1 296.052} C_DIS
LIN {X -0.079,Y -642.946,Z 1036.439,A 0.000,B 0.000,C 90.000,E1 295.079} C_DIS
LIN {X -0.136,Y -643.002,Z 1036.435,A 0.000,B 0.000,C 90.000,E1 294.335} C_DIS
LIN {X -0.118,Y -642.917,Z 1036.430,A 0.000,B 0.000,C 90.000,E1 293.334} C_DIS
LIN {X -0.042,Y -642.282,Z 1036.423,A 0.000,B 0.000,C 90.000,E1 292.078} C_DIS
LIN {X -0.161,Y -641.870,Z 1036.420,A 0.000,B 0.000,C 90.000,E1 291.589} C_DIS
LIN {X -0.281,Y -640.976,Z 1036.417,A 0.000,B 0.000,C 90.000,E1 291.099} C_DIS
LIN {X 0.370,Y -640.317,Z 1036.416,A 0.000,B 0.000,C 90.000,E1 290.791} C_DIS
LIN {X 0.240,Y -638.538,Z 1036.413,A 0.000,B 0.000,C 90.000,E1 290.301} C_DIS
LIN {X 0.262,Y -637.772,Z 1036.412,A 0.000,B 0.000,C 90.000,E1 290.174} C_DIS
LIN {X 0.139,Y -634.273,Z 1036.410,A 0.000,B 0.000,C 90.000,E1 289.704} C_DIS
LIN {X 0.155,Y -633.072,Z 1036.409,A 0.000,B 0.000,C 90.000,E1 289.577} C_DIS
LIN {X -0.195,Y -626.980,Z 1036.406,A 0.000,B 0.000,C 90.000,E1 289.141} C_DIS
LIN {X -0.189,Y -624.935,Z 1036.406,A 0.000,B 0.000,C 90.000,E1 289.033} C_DIS
LIN {X -0.243,Y -619.118,Z 1036.404,A 0.000,B 0.000,C 90.000,E1 288.779} C_DIS
LIN {X 0.192,Y -616.240,Z 1036.403,A 0.000,B 0.000,C 90.000,E1 288.598} C_DIS
LIN {X 0.279,Y -610.517,Z 1036.402,A 0.000,B 0.000,C 90.000,E1 288.362} C_DIS
LIN {X 0.098,Y -598.137,Z 1036.400,A 0.000,B 0.000,C 90.000,E1 287.946} C_DIS
LIN {X 0.243,Y -585.555,Z 1036.397,A 0.000,B 0.000,C 90.000,E1 287.511} C_DIS
LIN {X 0.033,Y -584.997,Z 1036.397,A 0.000,B 0.000,C 90.000,E1 287.511} C_DIS
LIN {X -0.003,Y -584.952,Z 1036.397,A 0.000,B 0.000,C 90.000,E1 287.511} C_DIS
LIN {X 0.062,Y -582.961,Z 1036.396,A 0.000,B 0.000,C 90.000,E1 287.347} C_DIS
LIN {X 0.088,Y -581.917,Z 1036.396,A 0.000,B 0.000,C 90.000,E1 287.330} C_DIS
LIN {X 0.038,Y -579.953,Z 1036.396,A 0.000,B 0.000,C 90.000,E1 287.330} C_DIS
LIN {X 0.007,Y -580.817,Z 1036.396,A 0.000,B 0.000,C 90.000,E1 287.275} C_DIS
LIN {X -0.202,Y -583.500,Z 1036.395,A 0.000,B 0.000,C 90.000,E1 287.040} C_DIS
LIN {X -0.107,Y -588.259,Z 1036.394,A 0.000,B 0.000,C 90.000,E1 286.913} C_DIS
LIN {X -0.162,Y -593.089,Z 1036.393,A 0.000,B 0.000,C 90.000,E1 286.677} C_DIS
LIN {X 0.027,Y -596.106,Z 1036.392,A 0.000,B 0.000,C 90.000,E1 286.496} C_DIS
LIN {X -0.145,Y -601.499,Z 1036.390,A 0.000,B 0.000,C 90.000,E1 286.134} C_DIS
LIN {X -0.114,Y -604.876,Z 1036.388,A 0.000,B 0.000,C 90.000,E1 285.788} C_DIS
LIN {X -0.174,Y -607.052,Z 1036.386,A 0.000,B 0.000,C 90.000,E1 285.536} C_DIS
LIN {X -0.114,Y -610.758,Z 1036.383,A 0.000,B 0.000,C 90.000,E1 285.009} C_DIS
LIN {X -0.025,Y -613.650,Z 1036.380,A 0.000,B 0.000,C 90.000,E1 284.481} C_DIS
LIN {X -0.071,Y -614.356,Z 1036.380,A 0.000,B 0.000,C 90.000,E1 284.356} C_DIS
LIN {X 0.283,Y -615.525,Z 1036.378,A 0.000,B 0.000,C 90.000,E1 284.064} C_DIS
LIN {X -0.193,Y -617.488,Z 1036.375,A 0.000,B 0.000,C 90.000,E1 283.592} C_DIS
LIN {X -0.055,Y -619.181,Z 1036.373,A 0.000,B 0.000,C 90.000,E1 283.063} C_DIS
LIN {X -0.283,Y -619.642,Z 1036.371,A 0.000,B 0.000,C 90.000,E1 282.827} C_DIS
LIN {X -0.128,Y -620.174,Z 1036.368,A 0.000,B 0.000,C 90.000,E1 282.299} C_DIS
LIN {X 0.031,Y -620.279,Z 1036.365,A 0.000,B 0.000,C 90.000,E1 281.771} C_DIS
LIN {X 0.191,Y -619.748,Z 1036.363,A 0.000,B 0.000,C 90.000,E1 281.243} C_DIS
LIN {X -0.035,Y -619.240,Z 1036.361,A 0.000,B 0.000,C 90.000,E1 281.007} C_DIS
LIN {X 0.002,Y -617.851,Z 1036.358,A 0.000,B 0.000,C 90.000,E1 280.489} C_DIS
LIN {X 0.144,Y -615.719,Z 1036.355,A 0.000,B 0.000,C 90.000,E1 279.962} C_DIS
LIN {X 0.164,Y -612.963,Z 1036.353,A 0.000,B 0.000,C 90.000,E1 279.443} C_DIS
LIN {X -0.085,Y -611.189,Z 1036.351,A 0.000,B 0.000,C 90.000,E1 279.208} C_DIS
LIN {X 0.171,Y -607.963,Z 1036.349,A 0.000,B 0.000,C 90.000,E1 278.803} C_DIS
LIN {X -0.218,Y -602.983,Z 1036.346,A 0.000,B 0.000,C 90.000,E1 278.341} C_DIS
LIN {X -0.227,Y -599.884,Z 1036.345,A 0.000,B 0.000,C 90.000,E1 278.106} C_DIS
LIN {X 0.176,Y -596.381,Z 1036.343,A 0.000,B 0.000,C 90.000,E1 277.757} C_DIS
LIN {X 0.037,Y -592.579,Z 1036.342,A 0.000,B 0.000,C 90.000,E1 277.530} C_DIS
LIN {X 0.061,Y -588.255,Z 1036.340,A 0.000,B 0.000,C 90.000,E1 277.239} C_DIS
LIN {X -0.044,Y -582.828,Z 1036.339,A 0.000,B 0.000,C 90.000,E1 277.004} C_DIS
LIN {X -0.234,Y -580.972,Z 1036.339,A 0.000,B 0.000,C 90.000,E1 276.947} C_DIS
LIN {X 0.237,Y -576.399,Z 1036.338,A 0.000,B 0.000,C 90.000,E1 276.777} C_DIS
LIN {X -0.250,Y -574.297,Z 1036.338,A 0.000,B 0.000,C 90.000,E1 276.777} C_DIS
LIN {X -0.059,Y -567.977,Z 1036.337,A 0.000,B 0.000,C 90.000,E1 276.720} C_DIS
LIN {X -0.087,Y -544.760,Z 1036.337,A 0.000,B 0.000,C 90.000,E1 276.720} C_DIS
LIN {X 0.096,Y -543.967,Z 1036.337,A 0.000,B 0.000,C 90.000,E1 276.606} C_DIS
LIN {X 0.054,Y -543.939,Z 1036.337,A 0.000,B 0.000,C 90.000,E1 276.606} C_DIS
LIN {X 0.156,Y -543.091,Z 1036.334,A 0.000,B 0.000,C 90.000,E1 276.087} C_DIS
LIN {X 0.139,Y -540.151,Z 1036.312,A 0.000,B 0.000,C 90.000,E1 272.121} C_DIS
LIN {X 0.230,Y -539.598,Z 1036.306,A 0.000,B 0.000,C 90.000,E1 270.974} C_DIS
LIN {X -0.239,Y -538.906,Z 1036.299,A 0.000,B 0.000,C 90.000,E1 269.885} C_DIS
LIN {X -0.168,Y -537.894,Z 1036.291,A 0.000,B 0.000,C 90.000,E1 268.453} C_DIS
LIN {X -0.073,Y -536.630,Z 1036.282,A 0.000,B 0.000,C 90.000,E1 266.731} C_DIS
LIN {X -0.034,Y -535.584,Z 1036.274,A 0.000,B 0.000,C 90.000,E1 265.298} C_DIS
LIN {X 0.070,Y -534.580,Z 1036.266,A 0.000,B 0.000,C 90.000,E1 263.856} C_DIS
LIN {X 0.120,Y -533.618,Z 1036.260,A 0.000,B 0.000,C 90.000,E1 262.704} C_DIS
LIN {X 0.222,Y -532.502,Z 1036.253,A 0.000,B 0.000,C 90.000,E1 261.546} C_DIS
LIN {X -0.216,Y -531.168,Z 1036.247,A 0.000,B 0.000,C 90.000,E1 260.443} C_DIS
LIN {X -0.086,Y -529.266,Z 1036.237,A 0.000,B 0.000,C 90.000,E1 258.701} C_DIS
LIN {X 0.210,Y -527.457,Z 1036.228,A 0.000,B 0.000,C 90.000,E1 256.937} C_DIS
LIN {X -0.028,Y -525.248,Z 1036.216,A 0.000,B 0.000,C 90.000,E1 254.936} C_DIS
LIN {X -0.056,Y -523.049,Z 1036.205,A 0.000,B 0.000,C 90.000,E1 252.906} C_DIS
LIN {X -0.114,Y -521.435,Z 1036.197,A 0.000,B 0.000,C 90.000,E1 251.456} C_DIS
LIN {X -0.059,Y -519.315,Z 1036.187,A 0.000,B 0.000,C 90.000,E1 249.699} C_DIS
LIN {X 0.121,Y -517.053,Z 1036.177,A 0.000,B 0.000,C 90.000,E1 247.922} C_DIS
LIN {X -0.162,Y -515.139,Z 1036.169,A 0.000,B 0.000,C 90.000,E1 246.485} C_DIS
LIN {X -0.253,Y -513.930,Z 1036.164,A 0.000,B 0.000,C 90.000,E1 245.613} C_DIS
LIN {X -0.045,Y -511.120,Z 1036.155,A 0.000,B 0.000,C 90.000,E1 243.819} C_DIS
LIN {X -0.222,Y -508.704,Z 1036.146,A 0.000,B 0.000,C 90.000,E1 242.359} C_DIS
LIN {X 0.026,Y -506.066,Z 1036.138,A 0.000,B 0.000,C 90.000,E1 240.845} C_DIS
LIN {X 0.227,Y -503.400,Z 1036.130,A 0.000,B 0.000,C 90.000,E1 239.331} C_DIS
LIN {X -0.061,Y -500.617,Z 1036.121,A 0.000,B 0.000,C 90.000,E1 237.867} C_DIS
LIN {X 0.266,Y -498.320,Z 1036.115,A 0.000,B 0.000,C 90.000,E1 236.628} C_DIS
LIN {X 0.003,Y -496.436,Z 1036.110,A 0.000,B 0.000,C 90.000,E1 235.754} C_DIS
LIN {X 0.000,Y -493.209,Z 1036.101,A 0.000,B 0.000,C 90.000,E1 234.242} C_DIS
LIN {X 0.047,Y -489.659,Z 1036.093,A 0.000,B 0.000,C 90.000,E1 232.718} C_DIS
LIN {X 0.051,Y -485.341,Z 1036.083,A 0.000,B 0.000,C 90.000,E1 230.884} C_DIS
LIN {X 0.194,Y -479.841,Z 1036.069,A 0.000,B 0.000,C 90.000,E1 228.405} C_DIS
LIN {X -0.106,Y -475.925,Z 1036.059,A 0.000,B 0.000,C 90.000,E1 226.581} C_DIS
LIN {X 0.276,Y -471.406,Z 1036.047,A 0.000,B 0.000,C 90.000,E1 224.352} C_DIS
LIN {X -0.136,Y -466.897,Z 1036.034,A 0.000,B 0.000,C 90.000,E1 222.204} C_DIS
LIN {X -0.088,Y -463.698,Z 1036.026,A 0.000,B 0.000,C 90.000,E1 220.620} C_DIS
LIN {X -0.001,Y -459.663,Z 1036.015,A 0.000,B 0.000,C 90.000,E1 218.705} C_DIS
LIN {X -0.018,Y -456.164,Z 1036.006,A 0.000,B 0.000,C 90.000,E1 217.111} C_DIS
LIN {X 0.038,Y -450.682,Z 1035.992,A 0.000,B 0.000,C 90.000,E1 214.532} C_DIS
LIN {X 0.001,Y -446.615,Z 1035.981,A 0.000,B 0.000,C 90.000,E1 212.594} C_DIS
LIN {X -0.229,Y -442.314,Z 1035.970,A 0.000,B 0.000,C 90.000,E1 210.669} C_DIS
LIN {X -0.031,Y -439.394,Z 1035.963,A 0.000,B 0.000,C 90.000,E1 209.333} C_DIS
LIN {X 0.133,Y -434.833,Z 1035.952,A 0.000,B 0.000,C 90.000,E1 207.334} C_DIS
LIN {X -0.198,Y -431.167,Z 1035.943,A 0.000,B 0.000,C 90.000,E1 205.720} C_DIS
LIN {X -0.042,Y -425.384,Z 1035.928,A 0.000,B 0.000,C 90.000,E1 203.025} C_DIS
LIN {X -0.017,Y -420.798,Z 1035.915,A 0.000,B 0.000,C 90.000,E1 200.663} C_DIS
LIN {X -0.171,Y -413.718,Z 1035.890,A 0.000,B 0.000,C 90.000,E1 196.260} C_DIS
LIN {X 0.025,Y -411.304,Z 1035.879,A 0.000,B 0.000,C 90.000,E1 194.175} C_DIS
LIN {X -0.151,Y -410.106,Z 1035.869,A 0.000,B 0.000,C 90.000,E1 192.479} C_DIS
LIN {X -0.038,Y -409.997,Z 1035.867,A 0.000,B 0.000,C 90.000,E1 192.119} C_DIS
LIN {X 0.040,Y -410.485,Z 1035.862,A 0.000,B 0.000,C 90.000,E1 191.074} C_DIS
LIN {X 0.069,Y -410.938,Z 1035.860,A 0.000,B 0.000,C 90.000,E1 190.725} C_DIS
LIN {X -0.121,Y -412.591,Z 1035.856,A 0.000,B 0.000,C 90.000,E1 190.074} C_DIS
LIN {X -0.139,Y -413.123,Z 1035.855,A 0.000,B 0.000,C 90.000,E1 189.905} C_DIS
LIN {X -0.048,Y -415.325,Z 1035.852,A 0.000,B 0.000,C 90.000,E1 189.378} C_DIS
LIN {X 0.094,Y -417.023,Z 1035.850,A 0.000,B 0.000,C 90.000,E1 189.029} C_DIS
LIN {X 0.146,Y -421.265,Z 1035.847,A 0.000,B 0.000,C 90.000,E1 188.341} C_DIS
LIN {X 0.087,Y -432.503,Z 1035.838,A 0.000,B 0.000,C 90.000,E1 186.834} C_DIS
LIN {X -0.159,Y -437.373,Z 1035.834,A 0.000,B 0.000,C 90.000,E1 186.201} C_DIS
LIN {X -0.025,Y -439.950,Z 1035.833,A 0.000,B 0.000,C 90.000,E1 185.853} C_DIS
LIN {X 0.032,Y -451.640,Z 1035.824,A 0.000,B 0.000,C 90.000,E1 184.302} C_DIS
LIN {X 0.084,Y -462.277,Z 1035.816,A 0.000,B 0.000,C 90.000,E1 182.865} C_DIS
LIN {X 0.121,Y -470.041,Z 1035.810,A 0.000,B 0.000,C 90.000,E1 181.776} C_DIS
LIN {X 0.053,Y -475.260,Z 1035.806,A 0.000,B 0.000,C 90.000,E1 181.031} C_DIS
LIN {X -0.146,Y -480.572,Z 1035.802,A 0.000,B 0.000,C 90.000,E1 180.286} C_DIS
LIN {X 0.009,Y -487.574,Z 1035.796,A 0.000,B 0.000,C 90.000,E1 179.198} C_DIS
LIN {X 0.006,Y -493.618,Z 1035.791,A 0.000,B 0.000,C 90.000,E1 178.282} C_DIS
LIN {X -0.230,Y -500.313,Z 1035.785,A 0.000,B 0.000,C 90.000,E1 177.249} C_DIS
LIN {X -0.013,Y -505.733,Z 1035.780,A 0.000,B 0.000,C 90.000,E1 176.331} C_DIS
LIN {X -0.066,Y -507.496,Z 1035.778,A 0.000,B 0.000,C 90.000,E1 176.045} C_DIS
LIN {X -0.176,Y -515.303,Z 1035.771,A 0.000,B 0.000,C 90.000,E1 174.723} C_DIS
LIN {X -0.162,Y -524.657,Z 1035.762,A 0.000,B 0.000,C 90.000,E1 173.109} C_DIS
LIN {X -0.136,Y -532.900,Z 1035.754,A 0.000,B 0.000,C 90.000,E1 171.659} C_DIS
LIN {X -0.225,Y -541.698,Z 1035.745,A 0.000,B 0.000,C 90.000,E1 170.095} C_DIS
LIN {X 0.220,Y -549.548,Z 1035.737,A 0.000,B 0.000,C 90.000,E1 168.634} C_DIS
LIN {X -0.248,Y -554.952,Z 1035.732,A 0.000,B 0.000,C 90.000,E1 167.701} C_DIS
LIN {X 0.146,Y -559.458,Z 1035.727,A 0.000,B 0.000,C 90.000,E1 166.825} C_DIS
LIN {X -0.215,Y -565.226,Z 1035.721,A 0.000,B 0.000,C 90.000,E1 165.755} C_DIS
LIN {X 0.060,Y -570.918,Z 1035.715,A 0.000,B 0.000,C 90.000,E1 164.629} C_DIS
LIN {X 0.318,Y -576.991,Z 1035.708,A 0.000,B 0.000,C 90.000,E1 163.378} C_DIS
LIN {X -0.270,Y -581.555,Z 1035.703,A 0.000,B 0.000,C 90.000,E1 162.489} C_DIS
LIN {X -0.238,Y -586.889,Z 1035.696,A 0.000,B 0.000,C 90.000,E1 161.275} C_DIS
LIN {X -0.058,Y -591.357,Z 1035.690,A 0.000,B 0.000,C 90.000,E1 160.188} C_DIS
LIN {X -0.168,Y -595.606,Z 1035.684,A 0.000,B 0.000,C 90.000,E1 159.135} C_DIS
LIN {X -0.122,Y -598.576,Z 1035.680,A 0.000,B 0.000,C 90.000,E1 158.337} C_DIS
LIN {X -0.123,Y -602.369,Z 1035.674,A 0.000,B 0.000,C 90.000,E1 157.283} C_DIS
LIN {X -0.075,Y -605.858,Z 1035.668,A 0.000,B 0.000,C 90.000,E1 156.230} C_DIS
LIN {X 0.012,Y -609.131,Z 1035.662,A 0.000,B 0.000,C 90.000,E1 155.177} C_DIS
LIN {X -0.193,Y -612.938,Z 1035.655,A 0.000,B 0.000,C 90.000,E1 153.896} C_DIS
LIN {X -0.330,Y -616.440,Z 1035.648,A 0.000,B 0.000,C 90.000,E1 152.615} C_DIS
LIN {X -0.122,Y -619.705,Z 1035.641,A 0.000,B 0.000,C 90.000,E1 151.307} C_DIS
LIN {X 0.149,Y -622.319,Z 1035.635,A 0.000,B 0.000,C 90.000,E1 150.255} C_DIS
LIN {X -0.080,Y -625.530,Z 1035.628,A 0.000,B 0.000,C 90.000,E1 148.997} C_DIS
LIN {X 0.075,Y -629.186,Z 1035.619,A 0.000,B 0.000,C 90.000,E1 147.454} C_DIS
LIN {X -0.247,Y -632.163,Z 1035.612,A 0.000,B 0.000,C 90.000,E1 146.215} C_DIS
LIN {X -0.146,Y -635.685,Z 1035.604,A 0.000,B 0.000,C 90.000,E1 144.689} C_DIS
LIN {X -0.107,Y -639.768,Z 1035.594,A 0.000,B 0.000,C 90.000,E1 142.924} C_DIS
LIN {X -0.013,Y -642.719,Z 1035.587,A 0.000,B 0.000,C 90.000,E1 141.662} C_DIS
LIN {X 0.071,Y -646.721,Z 1035.577,A 0.000,B 0.000,C 90.000,E1 139.908} C_DIS
LIN {X 0.161,Y -650.770,Z 1035.568,A 0.000,B 0.000,C 90.000,E1 138.162} C_DIS
LIN {X -0.223,Y -656.150,Z 1035.555,A 0.000,B 0.000,C 90.000,E1 135.972} C_DIS
LIN {X -0.020,Y -663.468,Z 1035.540,A 0.000,B 0.000,C 90.000,E1 133.257} C_DIS
LIN {X -0.067,Y -666.983,Z 1035.534,A 0.000,B 0.000,C 90.000,E1 132.043} C_DIS
LIN {X -0.019,Y -670.488,Z 1035.527,A 0.000,B 0.000,C 90.000,E1 130.825} C_DIS
LIN {X -0.349,Y -673.899,Z 1035.520,A 0.000,B 0.000,C 90.000,E1 129.644} C_DIS
LIN {X 0.331,Y -677.214,Z 1035.513,A 0.000,B 0.000,C 90.000,E1 128.382} C_DIS
LIN {X -0.305,Y -680.311,Z 1035.507,A 0.000,B 0.000,C 90.000,E1 127.237} C_DIS
LIN {X 0.061,Y -683.430,Z 1035.500,A 0.000,B 0.000,C 90.000,E1 126.011} C_DIS
LIN {X 0.074,Y -686.558,Z 1035.494,A 0.000,B 0.000,C 90.000,E1 124.818} C_DIS
LIN {X 0.341,Y -690.146,Z 1035.486,A 0.000,B 0.000,C 90.000,E1 123.372} C_DIS
LIN {X -0.280,Y -693.634,Z 1035.478,A 0.000,B 0.000,C 90.000,E1 122.005} C_DIS
LIN {X -0.151,Y -695.792,Z 1035.473,A 0.000,B 0.000,C 90.000,E1 121.052} C_DIS
LIN {X -0.353,Y -697.763,Z 1035.467,A 0.000,B 0.000,C 90.000,E1 120.129} C_DIS
LIN {X -0.184,Y -698.937,Z 1035.463,A 0.000,B 0.000,C 90.000,E1 119.411} C_DIS
LIN {X -0.077,Y -700.531,Z 1035.457,A 0.000,B 0.000,C 90.000,E1 118.231} C_DIS
LIN {X 0.006,Y -702.076,Z 1035.449,A 0.000,B 0.000,C 90.000,E1 116.821} C_DIS
LIN {X 0.216,Y -702.768,Z 1035.445,A 0.000,B 0.000,C 90.000,E1 116.104} C_DIS
LIN {X 0.049,Y -703.676,Z 1035.439,A 0.000,B 0.000,C 90.000,E1 114.951} C_DIS
LIN {X 0.036,Y -703.846,Z 1035.437,A 0.000,B 0.000,C 90.000,E1 114.719} C_DIS
LIN {X -0.039,Y -703.768,Z 1035.435,A 0.000,B 0.000,C 90.000,E1 114.259} C_DIS
LIN {X -0.045,Y -703.603,Z 1035.433,A 0.000,B 0.000,C 90.000,E1 114.027} C_DIS
LIN {X -0.127,Y -702.607,Z 1035.431,A 0.000,B 0.000,C 90.000,E1 113.567} C_DIS
LIN {X -0.130,Y -701.755,Z 1035.430,A 0.000,B 0.000,C 90.000,E1 113.334} C_DIS
LIN {X 0.141,Y -698.998,Z 1035.427,A 0.000,B 0.000,C 90.000,E1 112.845} C_DIS
LIN {X -0.370,Y -698.108,Z 1035.426,A 0.000,B 0.000,C 90.000,E1 112.770} C_DIS
LIN {X -0.239,Y -696.785,Z 1035.426,A 0.000,B 0.000,C 90.000,E1 112.642} C_DIS
LIN {X -0.252,Y -691.460,Z 1035.424,A 0.000,B 0.000,C 90.000,E1 112.333} C_DIS
LIN {X 0.230,Y -689.857,Z 1035.423,A 0.000,B 0.000,C 90.000,E1 112.206} C_DIS
LIN {X -0.141,Y -687.964,Z 1035.423,A 0.000,B 0.000,C 90.000,E1 112.153} C_DIS
LIN {X -0.252,Y -685.408,Z 1035.423,A 0.000,B 0.000,C 90.000,E1 112.078} C_DIS
LIN {X -0.290,Y -682.643,Z 1035.422,A 0.000,B 0.000,C 90.000,E1 112.025} C_DIS
LIN {X 0.220,Y -675.565,Z 1035.422,A 0.000,B 0.000,C 90.000,E1 111.897} C_DIS
LIN {X 0.153,Y -611.967,Z 1035.422,A 0.000,B 0.000,C 90.000,E1 111.897} C_DIS
LIN {X -0.181,Y -604.122,Z 1035.420,A 0.000,B 0.000,C 90.000,E1 111.663} C_DIS
LIN {X -0.211,Y -597.872,Z 1035.419,A 0.000,B 0.000,C 90.000,E1 111.354} C_DIS
LIN {X -0.067,Y -592.171,Z 1035.417,A 0.000,B 0.000,C 90.000,E1 110.972} C_DIS
LIN {X -0.010,Y -585.293,Z 1035.414,A 0.000,B 0.000,C 90.000,E1 110.429} C_DIS
LIN {X 0.207,Y -577.028,Z 1035.410,A 0.000,B 0.000,C 90.000,E1 109.704} C_DIS
LIN {X -0.013,Y -570.898,Z 1035.407,A 0.000,B 0.000,C 90.000,E1 109.268} C_DIS
LIN {X 0.162,Y -567.379,Z 1035.406,A 0.000,B 0.000,C 90.000,E1 109.033} C_DIS
LIN {X -0.083,Y -562.692,Z 1035.404,A 0.000,B 0.000,C 90.000,E1 108.779} C_DIS
LIN {X -0.170,Y -554.637,Z 1035.402,A 0.000,B 0.000,C 90.000,E1 108.362} C_DIS
LIN {X -0.071,Y -549.899,Z 1035.400,A 0.000,B 0.000,C 90.000,E1 108.055} C_DIS
LIN {X 0.124,Y -548.051,Z 1035.399,A 0.000,B 0.000,C 90.000,E1 107.819} C_DIS
LIN {X 0.083,Y -548.027,Z 1035.399,A 0.000,B 0.000,C 90.000,E1 107.819} C_DIS
LIN {X 0.169,Y -547.595,Z 1035.397,A 0.000,B 0.000,C 90.000,E1 107.511} C_DIS
LIN {X 0.206,Y -547.757,Z 1035.394,A 0.000,B 0.000,C 90.000,E1 106.804} C_DIS
LIN {X 0.113,Y -548.292,Z 1035.389,A 0.000,B 0.000,C 90.000,E1 105.969} C_DIS
LIN {X 0.146,Y -549.526,Z 1035.376,A 0.000,B 0.000,C 90.000,E1 103.716} C_DIS
LIN {X -0.001,Y -552.356,Z 1035.358,A 0.000,B 0.000,C 90.000,E1 100.366} C_DIS
LIN {X -0.190,Y -555.132,Z 1035.344,A 0.000,B 0.000,C 90.000,E1 97.871} C_DIS
LIN {X 0.286,Y -556.697,Z 1035.336,A 0.000,B 0.000,C 90.000,E1 96.429} C_DIS
LIN {X 0.183,Y -558.126,Z 1035.328,A 0.000,B 0.000,C 90.000,E1 95.049} C_DIS
LIN {X -0.096,Y -558.768,Z 1035.324,A 0.000,B 0.000,C 90.000,E1 94.245} C_DIS
LIN {X -0.251,Y -559.516,Z 1035.317,A 0.000,B 0.000,C 90.000,E1 93.151} C_DIS
LIN {X 0.213,Y -560.158,Z 1035.310,A 0.000,B 0.000,C 90.000,E1 91.718} C_DIS
LIN {X 0.024,Y -560.601,Z 1035.304,A 0.000,B 0.000,C 90.000,E1 90.630} C_DIS
LIN {X -0.059,Y -561.089,Z 1035.296,A 0.000,B 0.000,C 90.000,E1 89.255} C_DIS
LIN {X -0.024,Y -561.698,Z 1035.287,A 0.000,B 0.000,C 90.000,E1 87.593} C_DIS
LIN {X 0.056,Y -562.170,Z 1035.277,A 0.000,B 0.000,C 90.000,E1 85.927} C_DIS
LIN {X 0.054,Y -562.609,Z 1035.270,A 0.000,B 0.000,C 90.000,E1 84.546} C_DIS
LIN {X 0.053,Y -562.903,Z 1035.262,A 0.000,B 0.000,C 90.000,E1 83.166} C_DIS
LIN {X -0.059,Y -563.490,Z 1035.250,A 0.000,B 0.000,C 90.000,E1 80.971} C_DIS
LIN {X 0.188,Y -564.409,Z 1035.236,A 0.000,B 0.000,C 90.000,E1 78.465} C_DIS
LIN {X 0.157,Y -565.728,Z 1035.222,A 0.000,B 0.000,C 90.000,E1 75.992} C_DIS
LIN {X 0.146,Y -567.249,Z 1035.210,A 0.000,B 0.000,C 90.000,E1 73.795} C_DIS
LIN {X -0.167,Y -568.557,Z 1035.201,A 0.000,B 0.000,C 90.000,E1 72.181} C_DIS
LIN {X -0.287,Y -569.857,Z 1035.192,A 0.000,B 0.000,C 90.000,E1 70.550} C_DIS
LIN {X -0.009,Y -570.846,Z 1035.184,A 0.000,B 0.000,C 90.000,E1 69.156} C_DIS
LIN {X -0.218,Y -572.038,Z 1035.175,A 0.000,B 0.000,C 90.000,E1 67.539} C_DIS
LIN {X 0.126,Y -572.982,Z 1035.166,A 0.000,B 0.000,C 90.000,E1 65.869} C_DIS
LIN {X -0.326,Y -573.859,Z 1035.157,A 0.000,B 0.000,C 90.000,E1 64.280} C_DIS
LIN {X 0.012,Y -574.605,Z 1035.148,A 0.000,B 0.000,C 90.000,E1 62.615} C_DIS
LIN {X 0.007,Y -575.154,Z 1035.140,A 0.000,B 0.000,C 90.000,E1 61.257} C_DIS
LIN {X 0.128,Y -575.806,Z 1035.131,A 0.000,B 0.000,C 90.000,E1 59.616} C_DIS
LIN {X 0.083,Y -576.197,Z 1035.125,A 0.000,B 0.000,C 90.000,E1 58.535} C_DIS
LIN {X 0.192,Y -576.634,Z 1035.118,A 0.000,B 0.000,C 90.000,E1 57.168} C_DIS
LIN {X 0.160,Y -576.922,Z 1035.112,A 0.000,B 0.000,C 90.000,E1 56.087} C_DIS
LIN {X -0.025,Y -577.155,Z 1035.106,A 0.000,B 0.000,C 90.000,E1 55.022} C_DIS
LIN {X 0.084,Y -577.198,Z 1035.098,A 0.000,B 0.000,C 90.000,E1 53.657} C_DIS
LIN {X -0.051,Y -577.129,Z 1035.091,A 0.000,B 0.000,C 90.000,E1 52.316} C_DIS
LIN {X -0.235,Y -576.828,Z 1035.085,A 0.000,B 0.000,C 90.000,E1 51.251} C_DIS
LIN {X -0.214,Y -576.016,Z 1035.076,A 0.000,B 0.000,C 90.000,E1 49.622} C_DIS
LIN {X 0.018,Y -575.221,Z 1035.068,A 0.000,B 0.000,C 90.000,E1 48.243} C_DIS
LIN {X -0.188,Y -574.053,Z 1035.061,A 0.000,B 0.000,C 90.000,E1 46.905} C_DIS
LIN {X -0.119,Y -572.957,Z 1035.054,A 0.000,B 0.000,C 90.000,E1 45.810} C_DIS
LIN {X -0.078,Y -571.389,Z 1035.048,A 0.000,B 0.000,C 90.000,E1 44.717} C_DIS
LIN {X 0.244,Y -570.115,Z 1035.044,A 0.000,B 0.000,C 90.000,E1 43.866} C_DIS
LIN {X 0.253,Y -568.165,Z 1035.038,A 0.000,B 0.000,C 90.000,E1 42.771} C_DIS
LIN {X -0.254,Y -566.547,Z 1035.033,A 0.000,B 0.000,C 90.000,E1 42.000} C_DIS
LIN {X 0.023,Y -564.593,Z 1035.029,A 0.000,B 0.000,C 90.000,E1 41.148} C_DIS
LIN {X -0.091,Y -562.417,Z 1035.024,A 0.000,B 0.000,C 90.000,E1 40.334} C_DIS
LIN {X 0.132,Y -560.040,Z 1035.020,A 0.000,B 0.000,C 90.000,E1 39.483} C_DIS
LIN {X 0.225,Y -559.215,Z 1035.018,A 0.000,B 0.000,C 90.000,E1 39.197} C_DIS
LIN {X 0.136,Y -555.426,Z 1035.012,A 0.000,B 0.000,C 90.000,E1 38.096} C_DIS
LIN {X 0.290,Y -553.314,Z 1035.009,A 0.000,B 0.000,C 90.000,E1 37.523} C_DIS
LIN {X 0.052,Y -549.851,Z 1035.004,A 0.000,B 0.000,C 90.000,E1 36.710} C_DIS
LIN {X -0.108,Y -546.142,Z 1034.999,A 0.000,B 0.000,C 90.000,E1 35.884} C_DIS
LIN {X -0.024,Y -543.495,Z 1034.996,A 0.000,B 0.000,C 90.000,E1 35.311} C_DIS
LIN {X 0.058,Y -539.177,Z 1034.991,A 0.000,B 0.000,C 90.000,E1 34.452} C_DIS
LIN {X 0.083,Y -533.783,Z 1034.986,A 0.000,B 0.000,C 90.000,E1 33.452} C_DIS
LIN {X -0.085,Y -529.701,Z 1034.982,A 0.000,B 0.000,C 90.000,E1 32.752} C_DIS
LIN {X 0.149,Y -525.334,Z 1034.978,A 0.000,B 0.000,C 90.000,E1 32.005} C_DIS
LIN {X 0.175,Y -519.664,Z 1034.973,A 0.000,B 0.000,C 90.000,E1 31.131} C_DIS
LIN {X -0.056,Y -516.727,Z 1034.971,A 0.000,B 0.000,C 90.000,E1 30.718} C_DIS
LIN {X -0.035,Y -512.431,Z 1034.967,A 0.000,B 0.000,C 90.000,E1 30.129} C_DIS
LIN {X -0.043,Y -507.880,Z 1034.964,A 0.000,B 0.000,C 90.000,E1 29.539} C_DIS
LIN {X 0.101,Y -504.308,Z 1034.962,A 0.000,B 0.000,C 90.000,E1 29.077} C_DIS
LIN {X -0.204,Y -495.301,Z 1034.956,A 0.000,B 0.000,C 90.000,E1 28.103} C_DIS
LIN {X -0.142,Y -489.872,Z 1034.953,A 0.000,B 0.000,C 90.000,E1 27.513} C_DIS
LIN {X 0.168,Y -479.959,Z 1034.947,A 0.000,B 0.000,C 90.000,E1 26.488} C_DIS
LIN {X 0.104,Y -468.470,Z 1034.941,A 0.000,B 0.000,C 90.000,E1 25.412} C_DIS
LIN {X -0.144,Y -460.919,Z 1034.938,A 0.000,B 0.000,C 90.000,E1 24.771} C_DIS
LIN {X 0.200,Y -454.855,Z 1034.935,A 0.000,B 0.000,C 90.000,E1 24.207} C_DIS
LIN {X 0.013,Y -431.021,Z 1034.923,A 0.000,B 0.000,C 90.000,E1 22.153} C_DIS
LIN {X -0.088,Y -416.343,Z 1034.915,A 0.000,B 0.000,C 90.000,E1 20.737} C_DIS
LIN {X -0.136,Y -405.012,Z 1034.908,A 0.000,B 0.000,C 90.000,E1 19.504} C_DIS
LIN {X -0.060,Y -399.513,Z 1034.905,A 0.000,B 0.000,C 90.000,E1 18.833} C_DIS
LIN {X -0.072,Y -395.440,Z 1034.901,A 0.000,B 0.000,C 90.000,E1 18.236} C_DIS
LIN {X -0.079,Y -393.014,Z 1034.899,A 0.000,B 0.000,C 90.000,E1 17.764} C_DIS
LIN {X -0.061,Y -391.646,Z 1034.896,A 0.000,B 0.000,C 90.000,E1 17.221} C_DIS
LIN {X -0.221,Y -391.208,Z 1034.892,A 0.000,B 0.000,C 90.000,E1 16.622} C_DIS
LIN {X 0.045,Y -391.526,Z 1034.888,A 0.000,B 0.000,C 90.000,E1 15.843} C_DIS
LIN {X 0.043,Y -396.489,Z 1034.865,A 0.000,B 0.000,C 90.000,E1 11.591} C_DIS
LIN {X 0.171,Y -404.075,Z 1034.839,A 0.000,B 0.000,C 90.000,E1 7.011} C_DIS
LIN {X 0.122,Y -409.191,Z 1034.826,A 0.000,B 0.000,C 90.000,E1 4.588} C_DIS
LIN {X 0.096,Y -412.155,Z 1034.818,A 0.000,B 0.000,C 90.000,E1 3.212} C_DIS
LIN {X 0.113,Y -414.363,Z 1034.814,A 0.000,B 0.000,C 90.000,E1 2.522} C_DIS
LIN {X -0.067,Y -415.555,Z 1034.813,A 0.000,B 0.000,C 90.000,E1 2.293} C_DIS
LIN {X -0.044,Y -417.766,Z 1034.811,A 0.000,B 0.000,C 90.000,E1 1.892} C_DIS
LIN {X 0.035,Y -423.122,Z 1034.807,A 0.000,B 0.000,C 90.000,E1 1.318} C_DIS
LIN {X -0.179,Y -428.713,Z 1034.805,A 0.000,B 0.000,C 90.000,E1 0.974} C_DIS
LIN {X 0.207,Y -436.469,Z 1034.803,A 0.000,B 0.000,C 90.000,E1 0.458} C_DIS
LIN {X 0.008,Y -459.246,Z 1034.795,A 0.000,B 0.000,C 90.000,E1 359.083} C_DIS
LIN {X 0.143,Y -472.356,Z 1034.791,A 0.000,B 0.000,C 90.000,E1 358.282} C_DIS
LIN {X 0.111,Y -490.398,Z 1034.785,A 0.000,B 0.000,C 90.000,E1 357.192} C_DIS
LIN {X 0.108,Y -503.220,Z 1034.780,A 0.000,B 0.000,C 90.000,E1 356.388} C_DIS
LIN {X -0.229,Y -512.186,Z 1034.777,A 0.000,B 0.000,C 90.000,E1 355.812} C_DIS
LIN {X -0.121,Y -516.757,Z 1034.775,A 0.000,B 0.000,C 90.000,E1 355.469} C_DIS
LIN {X -0.005,Y -524.016,Z 1034.772,A 0.000,B 0.000,C 90.000,E1 354.894} C_DIS
LIN {X -0.252,Y -531.189,Z 1034.768,A 0.000,B 0.000,C 90.000,E1 354.318} C_DIS
LIN {X -0.068,Y -537.799,Z 1034.765,A 0.000,B 0.000,C 90.000,E1 353.685} C_DIS
LIN {X -0.164,Y -543.125,Z 1034.762,A 0.000,B 0.000,C 90.000,E1 353.166} C_DIS
LIN {X 0.092,Y -549.224,Z 1034.758,A 0.000,B 0.000,C 90.000,E1 352.470} C_DIS
LIN {X 0.106,Y -554.757,Z 1034.754,A 0.000,B 0.000,C 90.000,E1 351.781} C_DIS
LIN {X -0.194,Y -558.891,Z 1034.751,A 0.000,B 0.000,C 90.000,E1 351.254} C_DIS
LIN {X -0.152,Y -563.536,Z 1034.748,A 0.000,B 0.000,C 90.000,E1 350.557} C_DIS
LIN {X -0.069,Y -567.735,Z 1034.744,A 0.000,B 0.000,C 90.000,E1 349.859} C_DIS
LIN {X 0.050,Y -571.620,Z 1034.740,A 0.000,B 0.000,C 90.000,E1 349.162} C_DIS
LIN {X 0.080,Y -575.998,Z 1034.735,A 0.000,B 0.000,C 90.000,E1 348.342} C_DIS
LIN {X 0.156,Y -579.885,Z 1034.731,A 0.000,B 0.000,C 90.000,E1 347.521} C_DIS
LIN {X 0.036,Y -584.111,Z 1034.726,A 0.000,B 0.000,C 90.000,E1 346.589} C_DIS
LIN {X 0.006,Y -588.653,Z 1034.720,A 0.000,B 0.000,C 90.000,E1 345.519} C_DIS
LIN {X 0.044,Y -592.966,Z 1034.714,A 0.000,B 0.000,C 90.000,E1 344.448} C_DIS
LIN {X 0.142,Y -597.107,Z 1034.708,A 0.000,B 0.000,C 90.000,E1 343.378} C_DIS
LIN {X 0.009,Y -600.137,Z 1034.703,A 0.000,B 0.000,C 90.000,E1 342.598} C_DIS
LIN {X 0.192,Y -603.885,Z 1034.698,A 0.000,B 0.000,C 90.000,E1 341.529} C_DIS
LIN {X 0.038,Y -607.374,Z 1034.692,A 0.000,B 0.000,C 90.000,E1 340.496} C_DIS
LIN {X 0.144,Y -610.577,Z 1034.686,A 0.000,B 0.000,C 90.000,E1 339.444} C_DIS
LIN {X -0.225,Y -614.942,Z 1034.677,A 0.000,B 0.000,C 90.000,E1 337.922} C_DIS
LIN {X 0.254,Y -616.921,Z 1034.673,A 0.000,B 0.000,C 90.000,E1 337.102} C_DIS
LIN {X -0.065,Y -619.436,Z 1034.667,A 0.000,B 0.000,C 90.000,E1 336.102} C_DIS
LIN {X 0.206,Y -622.331,Z 1034.660,A 0.000,B 0.000,C 90.000,E1 334.793} C_DIS
LIN {X 0.222,Y -624.775,Z 1034.653,A 0.000,B 0.000,C 90.000,E1 333.512} C_DIS
LIN {X 0.281,Y -626.974,Z 1034.646,A 0.000,B 0.000,C 90.000,E1 332.231} C_DIS
LIN {X 0.118,Y -628.851,Z 1034.639,A 0.000,B 0.000,C 90.000,E1 330.973} C_DIS
LIN {X -0.322,Y -630.476,Z 1034.632,A 0.000,B 0.000,C 90.000,E1 329.744} C_DIS
LIN {X 0.413,Y -631.597,Z 1034.626,A 0.000,B 0.000,C 90.000,E1 328.663} C_DIS
LIN {X 0.298,Y -632.519,Z 1034.620,A 0.000,B 0.000,C 90.000,E1 327.661} C_DIS
LIN {X 0.023,Y -633.446,Z 1034.614,A 0.000,B 0.000,C 90.000,E1 326.421} C_DIS
LIN {X -0.099,Y -633.901,Z 1034.609,A 0.000,B 0.000,C 90.000,E1 325.674} C_DIS
LIN {X -0.370,Y -634.222,Z 1034.604,A 0.000,B 0.000,C 90.000,E1 324.689} C_DIS
LIN {X 0.121,Y -634.497,Z 1034.595,A 0.000,B 0.000,C 90.000,E1 323.130} C_DIS
LIN {X 0.367,Y -634.771,Z 1034.584,A 0.000,B 0.000,C 90.000,E1 321.090} C_DIS
LIN {X 0.376,Y -635.061,Z 1034.577,A 0.000,B 0.000,C 90.000,E1 319.828} C_DIS
LIN {X 0.278,Y -635.360,Z 1034.569,A 0.000,B 0.000,C 90.000,E1 318.324} C_DIS
LIN {X -0.029,Y -635.537,Z 1034.564,A 0.000,B 0.000,C 90.000,E1 317.595} C_DIS
LIN {X 0.203,Y -635.940,Z 1034.555,A 0.000,B 0.000,C 90.000,E1 315.810} C_DIS
LIN {X -0.380,Y -636.334,Z 1034.546,A 0.000,B 0.000,C 90.000,E1 314.352} C_DIS
LIN {X 0.131,Y -636.659,Z 1034.541,A 0.000,B 0.000,C 90.000,E1 313.299} C_DIS
LIN {X 0.107,Y -637.023,Z 1034.534,A 0.000,B 0.000,C 90.000,E1 312.043} C_DIS
LIN {X -0.062,Y -637.380,Z 1034.524,A 0.000,B 0.000,C 90.000,E1 310.297} C_DIS
LIN {X -0.017,Y -637.481,Z 1034.517,A 0.000,B 0.000,C 90.000,E1 309.036} C_DIS
LIN {X -0.206,Y -637.639,Z 1034.504,A 0.000,B 0.000,C 90.000,E1 306.790} C_DIS
LIN {X 0.160,Y -638.284,Z 1034.489,A 0.000,B 0.000,C 90.000,E1 303.992} C_DIS
LIN {X -0.040,Y -639.359,Z 1034.476,A 0.000,B 0.000,C 90.000,E1 301.750} C_DIS
LIN {X -0.163,Y -640.477,Z 1034.468,A 0.000,B 0.000,C 90.000,E1 300.256} C_DIS
LIN {X 0.087,Y -642.099,Z 1034.457,A 0.000,B 0.000,C 90.000,E1 298.231} C_DIS
LIN {X -0.206,Y -643.060,Z 1034.451,A 0.000,B 0.000,C 90.000,E1 297.257} C_DIS
LIN {X 0.086,Y -643.835,Z 1034.446,A 0.000,B 0.000,C 90.000,E1 296.232} C_DIS
LIN {X 0.311,Y -644.235,Z 1034.442,A 0.000,B 0.000,C 90.000,E1 295.463} C_DIS
LIN {X -0.321,Y -644.445,Z 1034.438,A 0.000,B 0.000,C 90.000,E1 294.771} C_DIS
LIN {X -0.283,Y -644.486,Z 1034.432,A 0.000,B 0.000,C 90.000,E1 293.770} C_DIS
LIN {X -0.066,Y -644.272,Z 1034.428,A 0.000,B 0.000,C 90.000,E1 293.003} C_DIS
LIN {X -0.285,Y -643.831,Z 1034.422,A 0.000,B 0.000,C 90.000,E1 292.025} C_DIS
LIN {X -0.392,Y -643.350,Z 1034.420,A 0.000,B 0.000,C 90.000,E1 291.535} C_DIS
LIN {X 0.329,Y -642.420,Z 1034.417,A 0.000,B 0.000,C 90.000,E1 290.972} C_DIS
LIN {X 0.158,Y -641.731,Z 1034.415,A 0.000,B 0.000,C 90.000,E1 290.737} C_DIS
LIN {X 0.213,Y -640.811,Z 1034.414,A 0.000,B 0.000,C 90.000,E1 290.482} C_DIS
LIN {X 0.041,Y -639.748,Z 1034.413,A 0.000,B 0.000,C 90.000,E1 290.248} C_DIS
LIN {X 0.064,Y -638.898,Z 1034.412,A 0.000,B 0.000,C 90.000,E1 290.120} C_DIS
LIN {X -0.110,Y -636.735,Z 1034.411,A 0.000,B 0.000,C 90.000,E1 289.885} C_DIS
LIN {X -0.076,Y -634.875,Z 1034.409,A 0.000,B 0.000,C 90.000,E1 289.631} C_DIS
LIN {X -0.061,Y -633.427,Z 1034.408,A 0.000,B 0.000,C 90.000,E1 289.504} C_DIS
LIN {X -0.079,Y -626.878,Z 1034.406,A 0.000,B 0.000,C 90.000,E1 289.033} C_DIS
LIN {X -0.193,Y -621.205,Z 1034.404,A 0.000,B 0.000,C 90.000,E1 288.779} C_DIS
LIN {X -0.178,Y -612.369,Z 1034.402,A 0.000,B 0.000,C 90.000,E1 288.417} C_DIS
LIN {X 0.299,Y -603.421,Z 1034.401,A 0.000,B 0.000,C 90.000,E1 288.055} C_DIS
LIN {X -0.126,Y -591.439,Z 1034.398,A 0.000,B 0.000,C 90.000,E1 287.692} C_DIS
LIN {X 0.029,Y -589.420,Z 1034.398,A 0.000,B 0.000,C 90.000,E1 287.583} C_DIS
LIN {X -0.024,Y -589.301,Z 1034.398,A 0.000,B 0.000,C 90.000,E1 287.583} C_DIS
LIN {X -0.094,Y -591.205,Z 1034.396,A 0.000,B 0.000,C 90.000,E1 287.330} C_DIS
LIN {X 0.033,Y -598.988,Z 1034.393,A 0.000,B 0.000,C 90.000,E1 286.804} C_DIS
LIN {X -0.233,Y -602.040,Z 1034.392,A 0.000,B 0.000,C 90.000,E1 286.622} C_DIS
LIN {X -0.239,Y -604.099,Z 1034.391,A 0.000,B 0.000,C 90.000,E1 286.441} C_DIS
LIN {X -0.258,Y -607.763,Z 1034.389,A 0.000,B 0.000,C 90.000,E1 286.079} C_DIS
LIN {X 0.072,Y -610.873,Z 1034.387,A 0.000,B 0.000,C 90.000,E1 285.662} C_DIS
LIN {X -0.227,Y -613.538,Z 1034.385,A 0.000,B 0.000,C 90.000,E1 285.300} C_DIS
LIN {X -0.120,Y -616.540,Z 1034.382,A 0.000,B 0.000,C 90.000,E1 284.773} C_DIS
LIN {X 0.202,Y -618.520,Z 1034.380,A 0.000,B 0.000,C 90.000,E1 284.356} C_DIS
LIN {X -0.255,Y -620.701,Z 1034.377,A 0.000,B 0.000,C 90.000,E1 283.883} C_DIS
LIN {X 0.124,Y -621.727,Z 1034.376,A 0.000,B 0.000,C 90.000,E1 283.592} C_DIS
LIN {X 0.292,Y -623.026,Z 1034.373,A 0.000,B 0.000,C 90.000,E1 283.063} C_DIS
LIN {X 0.077,Y -623.569,Z 1034.371,A 0.000,B 0.000,C 90.000,E1 282.827} C_DIS
LIN {X 0.260,Y -624.258,Z 1034.369,A 0.000,B 0.000,C 90.000,E1 282.299} C_DIS
LIN {X -0.163,Y -624.438,Z 1034.366,A 0.000,B 0.000,C 90.000,E1 281.827} C_DIS
LIN {X 0.236,Y -624.313,Z 1034.364,A 0.000,B 0.000,C 90.000,E1 281.535} C_DIS
LIN {X -0.309,Y -623.667,Z 1034.361,A 0.000,B 0.000,C 90.000,E1 281.074} C_DIS
LIN {X -0.124,Y -622.467,Z 1034.359,A 0.000,B 0.000,C 90.000,E1 280.546} C_DIS
LIN {X 0.050,Y -620.642,Z 1034.356,A 0.000,B 0.000,C 90.000,E1 280.018} C_DIS
LIN {X 0.269,Y -618.947,Z 1034.354,A 0.000,B 0.000,C 90.000,E1 279.613} C_DIS
LIN {X 0.038,Y -617.605,Z 1034.352,A 0.000,B 0.000,C 90.000,E1 279.378} C_DIS
LIN {X -0.098,Y -612.940,Z 1034.349,A 0.000,B 0.000,C 90.000,E1 278.746} C_DIS
LIN {X 0.083,Y -609.561,Z 1034.346,A 0.000,B 0.000,C 90.000,E1 278.341} C_DIS
LIN {X -0.210,Y -604.098,Z 1034.344,A 0.000,B 0.000,C 90.000,E1 277.871} C_DIS
LIN {X -0.265,Y -602.798,Z 1034.343,A 0.000,B 0.000,C 90.000,E1 277.757} C_DIS
LIN {X 0.151,Y -595.510,Z 1034.340,A 0.000,B 0.000,C 90.000,E1 277.182} C_DIS
LIN {X 0.253,Y -589.086,Z 1034.338,A 0.000,B 0.000,C 90.000,E1 276.777} C_DIS
LIN {X -0.137,Y -587.395,Z 1034.337,A 0.000,B 0.000,C 90.000,E1 276.720} C_DIS
LIN {X -0.159,Y -582.433,Z 1034.336,A 0.000,B 0.000,C 90.000,E1 276.543} C_DIS
LIN {X -0.175,Y -580.634,Z 1034.336,A 0.000,B 0.000,C 90.000,E1 276.486} C_DIS
LIN {X 0.163,Y -574.363,Z 1034.335,A 0.000,B 0.000,C 90.000,E1 276.315} C_DIS
LIN {X 0.053,Y -567.536,Z 1034.335,A 0.000,B 0.000,C 90.000,E1 276.258} C_DIS
LIN {X 0.016,Y -544.546,Z 1034.335,A 0.000,B 0.000,C 90.000,E1 276.258} C_DIS
LIN {X -0.019,Y -543.541,Z 1034.334,A 0.000,B 0.000,C 90.000,E1 276.087} C_DIS
LIN {X 0.090,Y -542.865,Z 1034.331,A 0.000,B 0.000,C 90.000,E1 275.625} C_DIS
LIN {X -0.033,Y -540.218,Z 1034.311,A 0.000,B 0.000,C 90.000,E1 271.949} C_DIS
LIN {X 0.077,Y -539.536,Z 1034.303,A 0.000,B 0.000,C 90.000,E1 270.516} C_DIS
LIN {X 0.161,Y -538.569,Z 1034.295,A 0.000,B 0.000,C 90.000,E1 269.083} C_DIS
LIN {X 0.248,Y -537.328,Z 1034.286,A 0.000,B 0.000,C 90.000,E1 267.364} C_DIS
LIN {X -0.238,Y -536.211,Z 1034.278,A 0.000,B 0.000,C 90.000,E1 265.988} C_DIS
LIN {X -0.090,Y -534.836,Z 1034.266,A 0.000,B 0.000,C 90.000,E1 263.970} C_DIS
LIN {X -0.057,Y -533.629,Z 1034.259,A 0.000,B 0.000,C 90.000,E1 262.534} C_DIS
LIN {X 0.075,Y -532.809,Z 1034.254,A 0.000,B 0.000,C 90.000,E1 261.659} C_DIS
LIN {X 0.169,Y -531.475,Z 1034.247,A 0.000,B 0.000,C 90.000,E1 260.500} C_DIS
LIN {X -0.176,Y -529.242,Z 1034.236,A 0.000,B 0.000,C 90.000,E1 258.522} C_DIS
LIN {X 0.125,Y -527.427,Z 1034.227,A 0.000,B 0.000,C 90.000,E1 256.756} C_DIS
LIN {X -0.111,Y -525.188,Z 1034.215,A 0.000,B 0.000,C 90.000,E1 254.755} C_DIS
LIN {X -0.134,Y -523.321,Z 1034.206,A 0.000,B 0.000,C 90.000,E1 253.015} C_DIS
LIN {X -0.194,Y -521.407,Z 1034.196,A 0.000,B 0.000,C 90.000,E1 251.275} C_DIS
LIN {X -0.107,Y -519.632,Z 1034.188,A 0.000,B 0.000,C 90.000,E1 249.806} C_DIS
LIN {X 0.091,Y -517.331,Z 1034.178,A 0.000,B 0.000,C 90.000,E1 248.028} C_DIS
LIN {X -0.253,Y -515.032,Z 1034.168,A 0.000,B 0.000,C 90.000,E1 246.305} C_DIS
LIN {X -0.135,Y -513.770,Z 1034.163,A 0.000,B 0.000,C 90.000,E1 245.409} C_DIS
LIN {X 0.203,Y -511.453,Z 1034.155,A 0.000,B 0.000,C 90.000,E1 243.896} C_DIS
LIN {X 0.026,Y -509.048,Z 1034.147,A 0.000,B 0.000,C 90.000,E1 242.436} C_DIS
LIN {X 0.275,Y -506.422,Z 1034.139,A 0.000,B 0.000,C 90.000,E1 240.923} C_DIS
LIN {X 0.042,Y -503.789,Z 1034.130,A 0.000,B 0.000,C 90.000,E1 239.459} C_DIS
LIN {X -0.110,Y -501.592,Z 1034.124,A 0.000,B 0.000,C 90.000,E1 238.280} C_DIS
LIN {X 0.101,Y -498.708,Z 1034.115,A 0.000,B 0.000,C 90.000,E1 236.755} C_DIS
LIN {X -0.016,Y -495.553,Z 1034.107,A 0.000,B 0.000,C 90.000,E1 235.261} C_DIS
LIN {X -0.176,Y -492.898,Z 1034.100,A 0.000,B 0.000,C 90.000,E1 234.069} C_DIS
LIN {X 0.288,Y -488.586,Z 1034.090,A 0.000,B 0.000,C 90.000,E1 232.190} C_DIS
LIN {X -0.064,Y -485.715,Z 1034.083,A 0.000,B 0.000,C 90.000,E1 231.009} C_DIS
LIN {X 0.103,Y -480.198,Z 1034.070,A 0.000,B 0.000,C 90.000,E1 228.528} C_DIS
LIN {X -0.161,Y -476.236,Z 1034.059,A 0.000,B 0.000,C 90.000,E1 226.701} C_DIS
LIN {X -0.112,Y -471.737,Z 1034.047,A 0.000,B 0.000,C 90.000,E1 224.514} C_DIS
LIN {X 0.076,Y -467.863,Z 1034.037,A 0.000,B 0.000,C 90.000,E1 222.609} C_DIS
LIN {X 0.202,Y -463.995,Z 1034.026,A 0.000,B 0.000,C 90.000,E1 220.701} C_DIS
LIN {X -0.063,Y -460.000,Z 1034.016,A 0.000,B 0.000,C 90.000,E1 218.830} C_DIS
LIN {X 0.185,Y -457.165,Z 1034.009,A 0.000,B 0.000,C 90.000,E1 217.523} C_DIS
LIN {X -0.250,Y -454.299,Z 1034.001,A 0.000,B 0.000,C 90.000,E1 216.297} C_DIS
LIN {X -0.021,Y -450.960,Z 1033.993,A 0.000,B 0.000,C 90.000,E1 214.659} C_DIS
LIN {X 0.080,Y -446.875,Z 1033.982,A 0.000,B 0.000,C 90.000,E1 212.704} C_DIS
LIN {X 0.100,Y -442.582,Z 1033.971,A 0.000,B 0.000,C 90.000,E1 210.747} C_DIS
LIN {X -0.079,Y -439.697,Z 1033.964,A 0.000,B 0.000,C 90.000,E1 209.461} C_DIS
LIN {X 0.091,Y -435.131,Z 1033.953,A 0.000,B 0.000,C 90.000,E1 207.462} C_DIS
LIN {X 0.154,Y -431.431,Z 1033.943,A 0.000,B 0.000,C 90.000,E1 205.796} C_DIS
LIN {X 0.130,Y -426.296,Z 1033.931,A 0.000,B 0.000,C 90.000,E1 203.462} C_DIS
LIN {X 0.182,Y -421.593,Z 1033.917,A 0.000,B 0.000,C 90.000,E1 201.099} C_DIS
LIN {X 0.112,Y -416.183,Z 1033.900,A 0.000,B 0.000,C 90.000,E1 198.055} C_DIS
LIN {X 0.053,Y -410.712,Z 1033.878,A 0.000,B 0.000,C 90.000,E1 193.953} C_DIS
LIN {X -0.060,Y -409.614,Z 1033.870,A 0.000,B 0.000,C 90.000,E1 192.591} C_DIS
LIN {X 0.096,Y -409.313,Z 1033.864,A 0.000,B 0.000,C 90.000,E1 191.535} C_DIS
LIN {X 0.142,Y -409.601,Z 1033.860,A 0.000,B 0.000,C 90.000,E1 190.838} C_DIS
LIN {X 0.168,Y -410.050,Z 1033.858,A 0.000,B 0.000,C 90.000,E1 190.489} C_DIS
LIN {X -0.127,Y -412.177,Z 1033.854,A 0.000,B 0.000,C 90.000,E1 189.670} C_DIS
LIN {X -0.109,Y -414.197,Z 1033.851,A 0.000,B 0.000,C 90.000,E1 189.208} C_DIS
LIN {X 0.081,Y -416.850,Z 1033.848,A 0.000,B 0.000,C 90.000,E1 188.681} C_DIS
LIN {X -0.191,Y -421.138,Z 1033.845,A 0.000,B 0.000,C 90.000,E1 188.049} C_DIS
LIN {X -0.177,Y -432.394,Z 1033.836,A 0.000,B 0.000,C 90.000,E1 186.543} C_DIS
LIN {X -0.115,Y -434.816,Z 1033.834,A 0.000,B 0.000,C 90.000,E1 186.201} C_DIS
LIN {X 0.050,Y -438.655,Z 1033.832,A 0.000,B 0.000,C 90.000,E1 185.682} C_DIS
LIN {X -0.033,Y -444.397,Z 1033.827,A 0.000,B 0.000,C 90.000,E1 184.935} C_DIS
LIN {X 0.192,Y -448.141,Z 1033.825,A 0.000,B 0.000,C 90.000,E1 184.416} C_DIS
LIN {X -0.189,Y -449.502,Z 1033.824,A 0.000,B 0.000,C 90.000,E1 184.302} C_DIS
LIN {X 0.069,Y -461.331,Z 1033.815,A 0.000,B 0.000,C 90.000,E1 182.694} C_DIS
LIN {X -0.194,Y -465.636,Z 1033.812,A 0.000,B 0.000,C 90.000,E1 182.121} C_DIS
LIN {X 0.042,Y -468.042,Z 1033.810,A 0.000,B 0.000,C 90.000,E1 181.776} C_DIS
LIN {X -0.045,Y -474.542,Z 1033.805,A 0.000,B 0.000,C 90.000,E1 180.859} C_DIS
LIN {X 0.148,Y -479.977,Z 1033.800,A 0.000,B 0.000,C 90.000,E1 180.057} C_DIS
LIN {X 0.218,Y -487.173,Z 1033.794,A 0.000,B 0.000,C 90.000,E1 178.969} C_DIS
LIN {X -0.094,Y -494.259,Z 1033.789,A 0.000,B 0.000,C 90.000,E1 177.936} C_DIS
LIN {X -0.026,Y -500.076,Z 1033.783,A 0.000,B 0.000,C 90.000,E1 177.020} C_DIS
LIN {X 0.168,Y -507.301,Z 1033.777,A 0.000,B 0.000,C 90.000,E1 175.812} C_DIS
LIN {X 0.109,Y -513.418,Z 1033.771,A 0.000,B 0.000,C 90.000,E1 174.780} C_DIS
LIN {X 0.199,Y -517.745,Z 1033.767,A 0.000,B 0.000,C 90.000,E1 174.033} C_DIS
LIN {X 0.091,Y -524.589,Z 1033.760,A 0.000,B 0.000,C 90.000,E1 172.875} C_DIS
LIN {X 0.049,Y -532.812,Z 1033.752,A 0.000,B 0.000,C 90.000,E1 171.432} C_DIS
LIN {X 0.229,Y -540.853,Z 1033.745,A 0.000,B 0.000,C 90.000,E1 169.982} C_DIS
LIN {X -0.151,Y -549.587,Z 1033.736,A 0.000,B 0.000,C 90.000,E1 168.465} C_DIS
LIN {X -0.087,Y -553.469,Z 1033.732,A 0.000,B 0.000,C 90.000,E1 167.757} C_DIS
LIN {X 0.153,Y -558.732,Z 1033.727,A 0.000,B 0.000,C 90.000,E1 166.756} C_DIS
LIN {X 0.075,Y -565.250,Z 1033.720,A 0.000,B 0.000,C 90.000,E1 165.519} C_DIS
LIN {X -0.199,Y -570.959,Z 1033.714,A 0.000,B 0.000,C 90.000,E1 164.448} C_DIS
LIN {X 0.059,Y -577.087,Z 1033.707,A 0.000,B 0.000,C 90.000,E1 163.196} C_DIS
LIN {X 0.285,Y -581.000,Z 1033.702,A 0.000,B 0.000,C 90.000,E1 162.362} C_DIS
LIN {X -0.161,Y -585.785,Z 1033.696,A 0.000,B 0.000,C 90.000,E1 161.329} C_DIS
LIN {X 0.009,Y -590.290,Z 1033.690,A 0.000,B 0.000,C 90.000,E1 160.242} C_DIS
LIN {X -0.324,Y -594.589,Z 1033.684,A 0.000,B 0.000,C 90.000,E1 159.209} C_DIS
LIN {X -0.293,Y -597.650,Z 1033.680,A 0.000,B 0.000,C 90.000,E1 158.411} C_DIS
LIN {X -0.315,Y -601.495,Z 1033.674,A 0.000,B 0.000,C 90.000,E1 157.358} C_DIS
LIN {X -0.285,Y -605.038,Z 1033.668,A 0.000,B 0.000,C 90.000,E1 156.305} C_DIS
LIN {X -0.011,Y -609.128,Z 1033.661,A 0.000,B 0.000,C 90.000,E1 154.973} C_DIS
LIN {X -0.173,Y -612.193,Z 1033.655,A 0.000,B 0.000,C 90.000,E1 153.948} C_DIS
LIN {X 0.230,Y -615.746,Z 1033.648,A 0.000,B 0.000,C 90.000,E1 152.615} C_DIS
LIN {X -0.126,Y -619.695,Z 1033.639,A 0.000,B 0.000,C 90.000,E1 151.101} C_DIS
LIN {X -0.155,Y -621.655,Z 1033.635,A 0.000,B 0.000,C 90.000,E1 150.333} C_DIS
LIN {X -0.079,Y -625.531,Z 1033.627,A 0.000,B 0.000,C 90.000,E1 148.791} C_DIS
LIN {X 0.078,Y -629.170,Z 1033.618,A 0.000,B 0.000,C 90.000,E1 147.248} C_DIS
LIN {X -0.244,Y -632.172,Z 1033.611,A 0.000,B 0.000,C 90.000,E1 146.008} C_DIS
LIN {X -0.145,Y -635.728,Z 1033.603,A 0.000,B 0.000,C 90.000,E1 144.482} C_DIS
LIN {X -0.117,Y -639.267,Z 1033.594,A 0.000,B 0.000,C 90.000,E1 142.970} C_DIS
LIN {X -0.014,Y -642.794,Z 1033.586,A 0.000,B 0.000,C 90.000,E1 141.457} C_DIS
LIN {X 0.141,Y -645.694,Z 1033.579,A 0.000,B 0.000,C 90.000,E1 140.194} C_DIS
LIN {X -0.217,Y -649.740,Z 1033.569,A 0.000,B 0.000,C 90.000,E1 138.485} C_DIS
LIN {X 0.247,Y -655.759,Z 1033.556,A 0.000,B 0.000,C 90.000,E1 135.972} C_DIS
LIN {X -0.004,Y -661.690,Z 1033.543,A 0.000,B 0.000,C 90.000,E1 133.785} C_DIS
LIN {X -0.048,Y -665.943,Z 1033.535,A 0.000,B 0.000,C 90.000,E1 132.324} C_DIS
LIN {X 0.437,Y -669.498,Z 1033.528,A 0.000,B 0.000,C 90.000,E1 131.067} C_DIS
LIN {X 0.097,Y -672.953,Z 1033.522,A 0.000,B 0.000,C 90.000,E1 129.886} C_DIS
LIN {X 0.243,Y -676.284,Z 1033.515,A 0.000,B 0.000,C 90.000,E1 128.669} C_DIS
LIN {X -0.011,Y -678.842,Z 1033.510,A 0.000,B 0.000,C 90.000,E1 127.729} C_DIS
LIN {X -0.059,Y -682.583,Z 1033.502,A 0.000,B 0.000,C 90.000,E1 126.297} C_DIS
LIN {X -0.044,Y -686.340,Z 1033.494,A 0.000,B 0.000,C 90.000,E1 124.865} C_DIS
LIN {X -0.171,Y -689.944,Z 1033.486,A 0.000,B 0.000,C 90.000,E1 123.452} C_DIS
LIN {X 0.163,Y -693.445,Z 1033.478,A 0.000,B 0.000,C 90.000,E1 122.005} C_DIS
LIN {X -0.067,Y -695.639,Z 1033.473,A 0.000,B 0.000,C 90.000,E1 121.082} C_DIS
LIN {X 0.087,Y -697.610,Z 1033.468,A 0.000,B 0.000,C 90.000,E1 120.129} C_DIS
LIN {X -0.090,Y -699.155,Z 1033.462,A 0.000,B 0.000,C 90.000,E1 119.205} C_DIS
LIN {X 0.363,Y -700.464,Z 1033.457,A 0.000,B 0.000,C 90.000,E1 118.231} C_DIS
LIN {X -0.109,Y -701.443,Z 1033.452,A 0.000,B 0.000,C 90.000,E1 117.334} C_DIS
LIN {X 0.375,Y -702.466,Z 1033.447,A 0.000,B 0.000,C 90.000,E1 116.360} C_DIS
LIN {X 0.206,Y -703.424,Z 1033.440,A 0.000,B 0.000,C 90.000,E1 115.207} C_DIS
LIN {X -0.166,Y -703.770,Z 1033.438,A 0.000,B 0.000,C 90.000,E1 114.771} C_DIS
LIN {X -0.251,Y -703.612,Z 1033.434,A 0.000,B 0.000,C 90.000,E1 114.079} C_DIS
LIN {X 0.028,Y -702.619,Z 1033.431,A 0.000,B 0.000,C 90.000,E1 113.590} C_DIS
LIN {X 0.306,Y -701.882,Z 1033.430,A 0.000,B 0.000,C 90.000,E1 113.334} C_DIS
LIN {X -0.069,Y -699.172,Z 1033.427,A 0.000,B 0.000,C 90.000,E1 112.898} C_DIS
LIN {X 0.064,Y -698.380,Z 1033.427,A 0.000,B 0.000,C 90.000,E1 112.770} C_DIS
LIN {X 0.194,Y -697.206,Z 1033.426,A 0.000,B 0.000,C 90.000,E1 112.642} C_DIS
LIN {X 0.192,Y -693.459,Z 1033.425,A 0.000,B 0.000,C 90.000,E1 112.408} C_DIS
LIN {X -0.132,Y -690.407,Z 1033.424,A 0.000,B 0.000,C 90.000,E1 112.259} C_DIS
LIN {X 0.112,Y -688.694,Z 1033.423,A 0.000,B 0.000,C 90.000,E1 112.153} C_DIS
LIN {X -0.080,Y -684.222,Z 1033.422,A 0.000,B 0.000,C 90.000,E1 112.025} C_DIS
LIN {X 0.117,Y -675.664,Z 1033.422,A 0.000,B 0.000,C 90.000,E1 111.897} C_DIS
LIN {X 0.046,Y -612.061,Z 1033.422,A 0.000,B 0.000,C 90.000,E1 111.897} C_DIS
LIN {X -0.213,Y -605.853,Z 1033.421,A 0.000,B 0.000,C 90.000,E1 111.716} C_DIS
LIN {X -0.058,Y -604.232,Z 1033.420,A 0.000,B 0.000,C 90.000,E1 111.642} C_DIS
LIN {X -0.158,Y -598.140,Z 1033.419,A 0.000,B 0.000,C 90.000,E1 111.354} C_DIS
LIN {X 0.244,Y -591.990,Z 1033.416,A 0.000,B 0.000,C 90.000,E1 110.918} C_DIS
LIN {X 0.084,Y -584.886,Z 1033.413,A 0.000,B 0.000,C 90.000,E1 110.375} C_DIS
LIN {X -0.053,Y -576.603,Z 1033.409,A 0.000,B 0.000,C 90.000,E1 109.685} C_DIS
LIN {X 0.081,Y -570.466,Z 1033.407,A 0.000,B 0.000,C 90.000,E1 109.214} C_DIS
LIN {X 0.036,Y -562.078,Z 1033.404,A 0.000,B 0.000,C 90.000,E1 108.725} C_DIS
LIN {X 0.238,Y -555.429,Z 1033.402,A 0.000,B 0.000,C 90.000,E1 108.362} C_DIS
LIN {X 0.144,Y -549.555,Z 1033.400,A 0.000,B 0.000,C 90.000,E1 108.000} C_DIS
LIN {X 0.146,Y -548.074,Z 1033.399,A 0.000,B 0.000,C 90.000,E1 107.819} C_DIS
LIN {X 0.104,Y -548.061,Z 1033.399,A 0.000,B 0.000,C 90.000,E1 107.819} C_DIS
LIN {X 0.152,Y -547.682,Z 1033.397,A 0.000,B 0.000,C 90.000,E1 107.528} C_DIS
LIN {X 0.077,Y -547.984,Z 1033.392,A 0.000,B 0.000,C 90.000,E1 106.551} C_DIS
LIN {X 0.075,Y -548.596,Z 1033.386,A 0.000,B 0.000,C 90.000,E1 105.426} C_DIS
LIN {X -0.003,Y -549.725,Z 1033.375,A 0.000,B 0.000,C 90.000,E1 103.467} C_DIS
LIN {X 0.151,Y -552.341,Z 1033.358,A 0.000,B 0.000,C 90.000,E1 100.366} C_DIS
LIN {X -0.282,Y -554.465,Z 1033.347,A 0.000,B 0.000,C 90.000,E1 98.454} C_DIS
LIN {X 0.189,Y -556.062,Z 1033.339,A 0.000,B 0.000,C 90.000,E1 97.011} C_DIS
LIN {X 0.139,Y -557.557,Z 1033.331,A 0.000,B 0.000,C 90.000,E1 95.625} C_DIS
LIN {X -0.023,Y -558.585,Z 1033.325,A 0.000,B 0.000,C 90.000,E1 94.531} C_DIS
LIN {X -0.129,Y -559.477,Z 1033.318,A 0.000,B 0.000,C 90.000,E1 93.154} C_DIS
LIN {X -0.195,Y -560.153,Z 1033.310,A 0.000,B 0.000,C 90.000,E1 91.776} C_DIS
LIN {X 0.270,Y -560.700,Z 1033.302,A 0.000,B 0.000,C 90.000,E1 90.344} C_DIS
LIN {X 0.188,Y -561.169,Z 1033.294,A 0.000,B 0.000,C 90.000,E1 88.969} C_DIS
LIN {X 0.127,Y -561.693,Z 1033.287,A 0.000,B 0.000,C 90.000,E1 87.593} C_DIS
LIN {X 0.075,Y -562.079,Z 1033.279,A 0.000,B 0.000,C 90.000,E1 86.216} C_DIS
LIN {X 0.152,Y -562.572,Z 1033.270,A 0.000,B 0.000,C 90.000,E1 84.552} C_DIS
LIN {X 0.204,Y -562.870,Z 1033.262,A 0.000,B 0.000,C 90.000,E1 83.166} C_DIS
LIN {X 0.091,Y -563.454,Z 1033.250,A 0.000,B 0.000,C 90.000,E1 80.971} C_DIS
LIN {X 0.173,Y -564.220,Z 1033.238,A 0.000,B 0.000,C 90.000,E1 78.757} C_DIS
LIN {X 0.223,Y -565.191,Z 1033.227,A 0.000,B 0.000,C 90.000,E1 76.825} C_DIS
LIN {X -0.127,Y -566.373,Z 1033.216,A 0.000,B 0.000,C 90.000,E1 74.936} C_DIS
LIN {X -0.138,Y -567.858,Z 1033.206,A 0.000,B 0.000,C 90.000,E1 73.015} C_DIS
LIN {X -0.104,Y -569.373,Z 1033.195,A 0.000,B 0.000,C 90.000,E1 71.094} C_DIS
LIN {X 0.170,Y -570.399,Z 1033.187,A 0.000,B 0.000,C 90.000,E1 69.699} C_DIS
LIN {X -0.074,Y -571.962,Z 1033.175,A 0.000,B 0.000,C 90.000,E1 67.539} C_DIS
LIN {X 0.103,Y -573.062,Z 1033.165,A 0.000,B 0.000,C 90.000,E1 65.613} C_DIS
LIN {X 0.171,Y -573.864,Z 1033.156,A 0.000,B 0.000,C 90.000,E1 63.973} C_DIS
LIN {X 0.150,Y -574.505,Z 1033.148,A 0.000,B 0.000,C 90.000,E1 62.615} C_DIS
LIN {X 0.144,Y -575.043,Z 1033.141,A 0.000,B 0.000,C 90.000,E1 61.257} C_DIS
LIN {X -0.234,Y -575.674,Z 1033.131,A 0.000,B 0.000,C 90.000,E1 59.665} C_DIS
LIN {X 0.215,Y -576.043,Z 1033.125,A 0.000,B 0.000,C 90.000,E1 58.535} C_DIS
LIN {X 0.010,Y -576.482,Z 1033.118,A 0.000,B 0.000,C 90.000,E1 57.199} C_DIS
LIN {X 0.288,Y -576.773,Z 1033.112,A 0.000,B 0.000,C 90.000,E1 56.087} C_DIS
LIN {X 0.101,Y -576.989,Z 1033.106,A 0.000,B 0.000,C 90.000,E1 55.022} C_DIS
LIN {X -0.258,Y -577.011,Z 1033.098,A 0.000,B 0.000,C 90.000,E1 53.703} C_DIS
LIN {X 0.069,Y -576.922,Z 1033.091,A 0.000,B 0.000,C 90.000,E1 52.316} C_DIS
LIN {X -0.118,Y -576.619,Z 1033.085,A 0.000,B 0.000,C 90.000,E1 51.251} C_DIS
LIN {X -0.102,Y -575.796,Z 1033.076,A 0.000,B 0.000,C 90.000,E1 49.622} C_DIS
LIN {X 0.125,Y -574.979,Z 1033.068,A 0.000,B 0.000,C 90.000,E1 48.243} C_DIS
LIN {X -0.085,Y -573.794,Z 1033.061,A 0.000,B 0.000,C 90.000,E1 46.905} C_DIS
LIN {X -0.021,Y -572.680,Z 1033.055,A 0.000,B 0.000,C 90.000,E1 45.810} C_DIS
LIN {X 0.017,Y -571.087,Z 1033.048,A 0.000,B 0.000,C 90.000,E1 44.717} C_DIS
LIN {X 0.335,Y -569.781,Z 1033.044,A 0.000,B 0.000,C 90.000,E1 43.866} C_DIS
LIN {X -0.077,Y -567.807,Z 1033.038,A 0.000,B 0.000,C 90.000,E1 42.813} C_DIS
LIN {X -0.171,Y -566.144,Z 1033.033,A 0.000,B 0.000,C 90.000,E1 42.000} C_DIS
LIN {X 0.101,Y -564.175,Z 1033.029,A 0.000,B 0.000,C 90.000,E1 41.148} C_DIS
LIN {X -0.019,Y -561.953,Z 1033.024,A 0.000,B 0.000,C 90.000,E1 40.334} C_DIS
LIN {X 0.107,Y -560.381,Z 1033.021,A 0.000,B 0.000,C 90.000,E1 39.769} C_DIS
LIN {X 0.291,Y -558.677,Z 1033.018,A 0.000,B 0.000,C 90.000,E1 39.197} C_DIS
LIN {X 0.193,Y -554.820,Z 1033.012,A 0.000,B 0.000,C 90.000,E1 38.096} C_DIS
LIN {X -0.027,Y -551.557,Z 1033.007,A 0.000,B 0.000,C 90.000,E1 37.282} C_DIS
LIN {X -0.120,Y -546.697,Z 1033.001,A 0.000,B 0.000,C 90.000,E1 36.171} C_DIS
LIN {X 0.007,Y -542.729,Z 1032.996,A 0.000,B 0.000,C 90.000,E1 35.311} C_DIS
LIN {X -0.081,Y -539.133,Z 1032.992,A 0.000,B 0.000,C 90.000,E1 34.612} C_DIS
LIN {X -0.349,Y -534.577,Z 1032.988,A 0.000,B 0.000,C 90.000,E1 33.785} C_DIS
LIN {X 0.072,Y -529.715,Z 1032.983,A 0.000,B 0.000,C 90.000,E1 32.880} C_DIS
LIN {X 0.306,Y -525.377,Z 1032.979,A 0.000,B 0.000,C 90.000,E1 32.133} C_DIS
LIN {X -0.222,Y -520.723,Z 1032.975,A 0.000,B 0.000,C 90.000,E1 31.465} C_DIS
LIN {X -0.073,Y -515.771,Z 1032.971,A 0.000,B 0.000,C 90.000,E1 30.718} C_DIS
LIN {X -0.058,Y -511.451,Z 1032.967,A 0.000,B 0.000,C 90.000,E1 30.129} C_DIS
LIN {X 0.106,Y -508.017,Z 1032.965,A 0.000,B 0.000,C 90.000,E1 29.667} C_DIS
LIN {X 0.064,Y -503.109,Z 1032.962,A 0.000,B 0.000,C 90.000,E1 29.077} C_DIS
LIN {X 0.139,Y -496.838,Z 1032.958,A 0.000,B 0.000,C 90.000,E1 28.359} C_DIS
LIN {X 0.269,Y -491.587,Z 1032.954,A 0.000,B 0.000,C 90.000,E1 27.769} C_DIS
LIN {X -0.003,Y -483.201,Z 1032.950,A 0.000,B 0.000,C 90.000,E1 26.950} C_DIS
LIN {X 0.243,Y -477.423,Z 1032.947,A 0.000,B 0.000,C 90.000,E1 26.360} C_DIS
LIN {X -0.216,Y -467.249,Z 1032.941,A 0.000,B 0.000,C 90.000,E1 25.463} C_DIS
LIN {X 0.069,Y -458.418,Z 1032.937,A 0.000,B 0.000,C 90.000,E1 24.643} C_DIS
LIN {X -0.123,Y -443.292,Z 1032.930,A 0.000,B 0.000,C 90.000,E1 23.387} C_DIS
LIN {X 0.196,Y -425.896,Z 1032.921,A 0.000,B 0.000,C 90.000,E1 21.770} C_DIS
LIN {X 0.141,Y -413.042,Z 1032.914,A 0.000,B 0.000,C 90.000,E1 20.482} C_DIS
LIN {X 0.153,Y -401.798,Z 1032.907,A 0.000,B 0.000,C 90.000,E1 19.214} C_DIS
LIN {X -0.029,Y -399.121,Z 1032.905,A 0.000,B 0.000,C 90.000,E1 18.906} C_DIS
LIN {X 0.163,Y -395.888,Z 1032.902,A 0.000,B 0.000,C 90.000,E1 18.417} C_DIS
LIN {X -0.103,Y -394.964,Z 1032.902,A 0.000,B 0.000,C 90.000,E1 18.290} C_DIS
LIN {X 0.124,Y -392.929,Z 1032.899,A 0.000,B 0.000,C 90.000,E1 17.819} C_DIS
LIN {X 0.085,Y -392.480,Z 1032.898,A 0.000,B 0.000,C 90.000,E1 17.692} C_DIS
LIN {X -0.097,Y -391.486,Z 1032.896,A 0.000,B 0.000,C 90.000,E1 17.275} C_DIS
LIN {X 0.118,Y -391.218,Z 1032.892,A 0.000,B 0.000,C 90.000,E1 16.622} C_DIS
LIN {X 0.146,Y -391.839,Z 1032.887,A 0.000,B 0.000,C 90.000,E1 15.552} C_DIS
LIN {X 0.189,Y -395.508,Z 1032.869,A 0.000,B 0.000,C 90.000,E1 12.355} C_DIS
LIN {X -0.014,Y -402.658,Z 1032.844,A 0.000,B 0.000,C 90.000,E1 7.814} C_DIS
LIN {X -0.156,Y -409.845,Z 1032.824,A 0.000,B 0.000,C 90.000,E1 4.359} C_DIS
LIN {X -0.166,Y -412.001,Z 1032.818,A 0.000,B 0.000,C 90.000,E1 3.326} C_DIS
LIN {X -0.124,Y -414.026,Z 1032.815,A 0.000,B 0.000,C 90.000,E1 2.636} C_DIS
LIN {X -0.116,Y -416.272,Z 1032.812,A 0.000,B 0.000,C 90.000,E1 2.121} C_DIS
LIN {X -0.111,Y -417.171,Z 1032.811,A 0.000,B 0.000,C 90.000,E1 1.949} C_DIS
LIN {X 0.168,Y -418.131,Z 1032.810,A 0.000,B 0.000,C 90.000,E1 1.776} C_DIS
LIN {X 0.115,Y -422.943,Z 1032.807,A 0.000,B 0.000,C 90.000,E1 1.260} C_DIS
LIN {X 0.048,Y -428.062,Z 1032.805,A 0.000,B 0.000,C 90.000,E1 0.917} C_DIS
LIN {X -0.164,Y -433.493,Z 1032.803,A 0.000,B 0.000,C 90.000,E1 0.630} C_DIS
LIN {X -0.079,Y -449.895,Z 1032.798,A 0.000,B 0.000,C 90.000,E1 359.599} C_DIS
LIN {X 0.222,Y -466.473,Z 1032.792,A 0.000,B 0.000,C 90.000,E1 358.568} C_DIS
LIN {X -0.067,Y -474.645,Z 1032.790,A 0.000,B 0.000,C 90.000,E1 358.108} C_DIS
LIN {X -0.204,Y -491.067,Z 1032.784,A 0.000,B 0.000,C 90.000,E1 357.135} C_DIS
LIN {X 0.158,Y -500.514,Z 1032.781,A 0.000,B 0.000,C 90.000,E1 356.502} C_DIS
LIN {X 0.210,Y -510.024,Z 1032.777,A 0.000,B 0.000,C 90.000,E1 355.869} C_DIS
LIN {X -0.112,Y -516.136,Z 1032.775,A 0.000,B 0.000,C 90.000,E1 355.469} C_DIS
LIN {X 0.063,Y -523.411,Z 1032.772,A 0.000,B 0.000,C 90.000,E1 354.894} C_DIS
LIN {X -0.115,Y -530.545,Z 1032.768,A 0.000,B 0.000,C 90.000,E1 354.318} C_DIS
LIN {X -0.001,Y -538.511,Z 1032.764,A 0.000,B 0.000,C 90.000,E1 353.571} C_DIS
LIN {X -0.071,Y -543.781,Z 1032.761,A 0.000,B 0.000,C 90.000,E1 353.053} C_DIS
LIN {X -0.152,Y -548.714,Z 1032.758,A 0.000,B 0.000,C 90.000,E1 352.527} C_DIS
LIN {X -0.140,Y -554.291,Z 1032.755,A 0.000,B 0.000,C 90.000,E1 351.837} C_DIS
LIN {X 0.108,Y -558.533,Z 1032.751,A 0.000,B 0.000,C 90.000,E1 351.254} C_DIS
LIN {X 0.149,Y -563.208,Z 1032.748,A 0.000,B 0.000,C 90.000,E1 350.557} C_DIS
LIN {X -0.182,Y -566.675,Z 1032.745,A 0.000,B 0.000,C 90.000,E1 350.038} C_DIS
LIN {X -0.076,Y -570.681,Z 1032.741,A 0.000,B 0.000,C 90.000,E1 349.342} C_DIS
LIN {X 0.178,Y -574.423,Z 1032.737,A 0.000,B 0.000,C 90.000,E1 348.634} C_DIS
LIN {X -0.093,Y -577.179,Z 1032.734,A 0.000,B 0.000,C 90.000,E1 348.117} C_DIS
LIN {X -0.120,Y -581.634,Z 1032.729,A 0.000,B 0.000,C 90.000,E1 347.173} C_DIS
LIN {X 0.009,Y -585.213,Z 1032.724,A 0.000,B 0.000,C 90.000,E1 346.353} C_DIS
LIN {X 0.313,Y -588.663,Z 1032.720,A 0.000,B 0.000,C 90.000,E1 345.519} C_DIS
LIN {X 0.046,Y -594.053,Z 1032.712,A 0.000,B 0.000,C 90.000,E1 344.212} C_DIS
LIN {X -0.136,Y -599.227,Z 1032.705,A 0.000,B 0.000,C 90.000,E1 342.906} C_DIS
LIN {X -0.255,Y -602.161,Z 1032.701,A 0.000,B 0.000,C 90.000,E1 342.127} C_DIS
LIN {X 0.142,Y -605.795,Z 1032.695,A 0.000,B 0.000,C 90.000,E1 341.040} C_DIS
LIN {X 0.016,Y -609.174,Z 1032.689,A 0.000,B 0.000,C 90.000,E1 340.007} C_DIS
LIN {X 0.200,Y -611.518,Z 1032.685,A 0.000,B 0.000,C 90.000,E1 339.209} C_DIS
LIN {X 0.073,Y -615.877,Z 1032.676,A 0.000,B 0.000,C 90.000,E1 337.667} C_DIS
LIN {X 0.287,Y -619.114,Z 1032.669,A 0.000,B 0.000,C 90.000,E1 336.357} C_DIS
LIN {X -0.011,Y -622.058,Z 1032.662,A 0.000,B 0.000,C 90.000,E1 335.101} C_DIS
LIN {X -0.009,Y -623.643,Z 1032.657,A 0.000,B 0.000,C 90.000,E1 334.332} C_DIS
LIN {X 0.026,Y -625.578,Z 1032.652,A 0.000,B 0.000,C 90.000,E1 333.307} C_DIS
LIN {X 0.084,Y -627.388,Z 1032.646,A 0.000,B 0.000,C 90.000,E1 332.281} C_DIS
LIN {X 0.179,Y -629.288,Z 1032.639,A 0.000,B 0.000,C 90.000,E1 331.001} C_DIS
LIN {X 0.053,Y -630.959,Z 1032.632,A 0.000,B 0.000,C 90.000,E1 329.744} C_DIS
LIN {X 0.281,Y -632.356,Z 1032.625,A 0.000,B 0.000,C 90.000,E1 328.456} C_DIS
LIN {X -0.335,Y -633.477,Z 1032.618,A 0.000,B 0.000,C 90.000,E1 327.248} C_DIS
LIN {X -0.067,Y -634.388,Z 1032.611,A 0.000,B 0.000,C 90.000,E1 325.960} C_DIS
LIN {X -0.333,Y -634.840,Z 1032.605,A 0.000,B 0.000,C 90.000,E1 324.975} C_DIS
LIN {X 0.169,Y -635.184,Z 1032.597,A 0.000,B 0.000,C 90.000,E1 323.417} C_DIS
LIN {X -0.211,Y -635.339,Z 1032.590,A 0.000,B 0.000,C 90.000,E1 322.190} C_DIS
LIN {X 0.051,Y -635.788,Z 1032.579,A 0.000,B 0.000,C 90.000,E1 320.150} C_DIS
LIN {X -0.039,Y -636.109,Z 1032.570,A 0.000,B 0.000,C 90.000,E1 318.647} C_DIS
LIN {X 0.027,Y -636.394,Z 1032.565,A 0.000,B 0.000,C 90.000,E1 317.634} C_DIS
LIN {X -0.192,Y -636.836,Z 1032.555,A 0.000,B 0.000,C 90.000,E1 315.891} C_DIS
LIN {X 0.142,Y -637.277,Z 1032.547,A 0.000,B 0.000,C 90.000,E1 314.352} C_DIS
LIN {X -0.234,Y -637.602,Z 1032.541,A 0.000,B 0.000,C 90.000,E1 313.380} C_DIS
LIN {X -0.051,Y -637.859,Z 1032.537,A 0.000,B 0.000,C 90.000,E1 312.609} C_DIS
LIN {X 0.137,Y -638.076,Z 1032.533,A 0.000,B 0.000,C 90.000,E1 311.838} C_DIS
LIN {X 0.102,Y -638.439,Z 1032.524,A 0.000,B 0.000,C 90.000,E1 310.334} C_DIS
LIN {X -0.319,Y -638.588,Z 1032.517,A 0.000,B 0.000,C 90.000,E1 309.116} C_DIS
LIN {X -0.253,Y -638.670,Z 1032.509,A 0.000,B 0.000,C 90.000,E1 307.604} C_DIS
LIN {X -0.180,Y -638.864,Z 1032.500,A 0.000,B 0.000,C 90.000,E1 306.091} C_DIS
LIN {X -0.191,Y -639.546,Z 1032.488,A 0.000,B 0.000,C 90.000,E1 303.833} C_DIS
LIN {X -0.308,Y -641.647,Z 1032.468,A 0.000,B 0.000,C 90.000,E1 300.335} C_DIS
LIN {X 0.267,Y -642.479,Z 1032.463,A 0.000,B 0.000,C 90.000,E1 299.283} C_DIS
LIN {X 0.007,Y -644.354,Z 1032.452,A 0.000,B 0.000,C 90.000,E1 297.308} C_DIS
LIN {X 0.025,Y -645.173,Z 1032.446,A 0.000,B 0.000,C 90.000,E1 296.309} C_DIS
LIN {X -0.235,Y -645.756,Z 1032.441,A 0.000,B 0.000,C 90.000,E1 295.335} C_DIS
LIN {X -0.184,Y -645.964,Z 1032.435,A 0.000,B 0.000,C 90.000,E1 294.335} C_DIS
LIN {X 0.053,Y -645.957,Z 1032.431,A 0.000,B 0.000,C 90.000,E1 293.567} C_DIS
LIN {X 0.029,Y -645.715,Z 1032.427,A 0.000,B 0.000,C 90.000,E1 292.823} C_DIS
LIN {X 0.001,Y -645.496,Z 1032.423,A 0.000,B 0.000,C 90.000,E1 292.078} C_DIS
LIN {X -0.098,Y -645.007,Z 1032.420,A 0.000,B 0.000,C 90.000,E1 291.589} C_DIS
LIN {X -0.197,Y -644.158,Z 1032.417,A 0.000,B 0.000,C 90.000,E1 291.099} C_DIS
LIN {X -0.134,Y -643.653,Z 1032.416,A 0.000,B 0.000,C 90.000,E1 290.844} C_DIS
LIN {X 0.164,Y -641.102,Z 1032.412,A 0.000,B 0.000,C 90.000,E1 290.194} C_DIS
LIN {X 0.191,Y -640.258,Z 1032.412,A 0.000,B 0.000,C 90.000,E1 290.066} C_DIS
LIN {X 0.040,Y -636.882,Z 1032.410,A 0.000,B 0.000,C 90.000,E1 289.704} C_DIS
LIN {X 0.060,Y -635.896,Z 1032.409,A 0.000,B 0.000,C 90.000,E1 289.577} C_DIS
LIN {X 0.075,Y -634.420,Z 1032.408,A 0.000,B 0.000,C 90.000,E1 289.450} C_DIS
LIN {X 0.232,Y -630.723,Z 1032.407,A 0.000,B 0.000,C 90.000,E1 289.214} C_DIS
LIN {X -0.109,Y -627.858,Z 1032.406,A 0.000,B 0.000,C 90.000,E1 289.033} C_DIS
LIN {X 0.354,Y -623.459,Z 1032.405,A 0.000,B 0.000,C 90.000,E1 288.779} C_DIS
LIN {X 0.361,Y -614.851,Z 1032.403,A 0.000,B 0.000,C 90.000,E1 288.417} C_DIS
LIN {X 0.155,Y -604.217,Z 1032.400,A 0.000,B 0.000,C 90.000,E1 288.055} C_DIS
LIN {X 0.301,Y -593.939,Z 1032.399,A 0.000,B 0.000,C 90.000,E1 287.692} C_DIS
LIN {X 0.261,Y -593.955,Z 1032.398,A 0.000,B 0.000,C 90.000,E1 287.692} C_DIS
LIN {X 0.086,Y -597.037,Z 1032.397,A 0.000,B 0.000,C 90.000,E1 287.457} C_DIS
LIN {X 0.138,Y -599.642,Z 1032.396,A 0.000,B 0.000,C 90.000,E1 287.221} C_DIS
LIN {X 0.278,Y -603.496,Z 1032.394,A 0.000,B 0.000,C 90.000,E1 286.913} C_DIS
LIN {X -0.176,Y -608.771,Z 1032.392,A 0.000,B 0.000,C 90.000,E1 286.496} C_DIS
LIN {X -0.256,Y -609.936,Z 1032.391,A 0.000,B 0.000,C 90.000,E1 286.386} C_DIS
LIN {X 0.026,Y -614.865,Z 1032.387,A 0.000,B 0.000,C 90.000,E1 285.717} C_DIS
LIN {X 0.105,Y -618.837,Z 1032.384,A 0.000,B 0.000,C 90.000,E1 285.064} C_DIS
LIN {X 0.251,Y -621.476,Z 1032.381,A 0.000,B 0.000,C 90.000,E1 284.537} C_DIS
LIN {X 0.031,Y -622.751,Z 1032.380,A 0.000,B 0.000,C 90.000,E1 284.300} C_DIS
LIN {X -0.186,Y -623.809,Z 1032.378,A 0.000,B 0.000,C 90.000,E1 284.064} C_DIS
LIN {X -0.005,Y -625.452,Z 1032.375,A 0.000,B 0.000,C 90.000,E1 283.536} C_DIS
LIN {X 0.192,Y -626.879,Z 1032.372,A 0.000,B 0.000,C 90.000,E1 283.008} C_DIS
LIN {X -0.011,Y -627.360,Z 1032.371,A 0.000,B 0.000,C 90.000,E1 282.771} C_DIS
LIN {X 0.199,Y -627.827,Z 1032.368,A 0.000,B 0.000,C 90.000,E1 282.243} C_DIS
LIN {X -0.201,Y -627.919,Z 1032.365,A 0.000,B 0.000,C 90.000,E1 281.771} C_DIS
LIN {X 0.213,Y -627.805,Z 1032.364,A 0.000,B 0.000,C 90.000,E1 281.478} C_DIS
LIN {X -0.191,Y -627.274,Z 1032.361,A 0.000,B 0.000,C 90.000,E1 281.007} C_DIS
LIN {X -0.100,Y -626.178,Z 1032.358,A 0.000,B 0.000,C 90.000,E1 280.489} C_DIS
LIN {X 0.101,Y -624.377,Z 1032.355,A 0.000,B 0.000,C 90.000,E1 279.962} C_DIS
LIN {X 0.182,Y -622.122,Z 1032.353,A 0.000,B 0.000,C 90.000,E1 279.443} C_DIS
LIN {X 0.122,Y -621.536,Z 1032.352,A 0.000,B 0.000,C 90.000,E1 279.321} C_DIS
LIN {X 0.114,Y -617.539,Z 1032.348,A 0.000,B 0.000,C 90.000,E1 278.681} C_DIS
LIN {X 0.147,Y -613.073,Z 1032.345,A 0.000,B 0.000,C 90.000,E1 278.163} C_DIS
LIN {X -0.125,Y -609.365,Z 1032.343,A 0.000,B 0.000,C 90.000,E1 277.814} C_DIS
LIN {X -0.216,Y -606.639,Z 1032.342,A 0.000,B 0.000,C 90.000,E1 277.587} C_DIS
LIN {X -0.141,Y -600.852,Z 1032.340,A 0.000,B 0.000,C 90.000,E1 277.125} C_DIS
LIN {X -0.102,Y -593.048,Z 1032.337,A 0.000,B 0.000,C 90.000,E1 276.606} C_DIS
LIN {X 0.104,Y -587.897,Z 1032.335,A 0.000,B 0.000,C 90.000,E1 276.315} C_DIS
LIN {X 0.249,Y -580.345,Z 1032.334,A 0.000,B 0.000,C 90.000,E1 276.030} C_DIS
LIN {X 0.164,Y -573.549,Z 1032.333,A 0.000,B 0.000,C 90.000,E1 275.910} C_DIS
LIN {X 0.146,Y -567.189,Z 1032.333,A 0.000,B 0.000,C 90.000,E1 275.853} C_DIS
LIN {X 0.086,Y -543.970,Z 1032.333,A 0.000,B 0.000,C 90.000,E1 275.853} C_DIS
LIN {X 0.235,Y -543.124,Z 1032.330,A 0.000,B 0.000,C 90.000,E1 275.454} C_DIS
LIN {X -0.049,Y -541.467,Z 1032.321,A 0.000,B 0.000,C 90.000,E1 273.784} C_DIS
LIN {X 0.198,Y -539.931,Z 1032.305,A 0.000,B 0.000,C 90.000,E1 270.917} C_DIS
LIN {X -0.266,Y -539.253,Z 1032.299,A 0.000,B 0.000,C 90.000,E1 269.828} C_DIS
LIN {X -0.161,Y -538.038,Z 1032.289,A 0.000,B 0.000,C 90.000,E1 268.108} C_DIS
LIN {X -0.122,Y -537.185,Z 1032.283,A 0.000,B 0.000,C 90.000,E1 266.963} C_DIS
LIN {X -0.011,Y -535.482,Z 1032.270,A 0.000,B 0.000,C 90.000,E1 264.666} C_DIS
LIN {X 0.049,Y -534.657,Z 1032.264,A 0.000,B 0.000,C 90.000,E1 263.514} C_DIS
LIN {X 0.209,Y -533.417,Z 1032.256,A 0.000,B 0.000,C 90.000,E1 262.064} C_DIS
LIN {X 0.267,Y -532.530,Z 1032.251,A 0.000,B 0.000,C 90.000,E1 261.197} C_DIS
LIN {X 0.026,Y -529.549,Z 1032.237,A 0.000,B 0.000,C 90.000,E1 258.634} C_DIS
LIN {X 0.221,Y -527.754,Z 1032.227,A 0.000,B 0.000,C 90.000,E1 256.881} C_DIS
LIN {X 0.121,Y -525.529,Z 1032.216,A 0.000,B 0.000,C 90.000,E1 254.866} C_DIS
LIN {X -0.040,Y -523.320,Z 1032.205,A 0.000,B 0.000,C 90.000,E1 252.851} C_DIS
LIN {X -0.099,Y -521.764,Z 1032.197,A 0.000,B 0.000,C 90.000,E1 251.402} C_DIS
LIN {X -0.042,Y -519.587,Z 1032.187,A 0.000,B 0.000,C 90.000,E1 249.645} C_DIS
LIN {X -0.147,Y -517.258,Z 1032.177,A 0.000,B 0.000,C 90.000,E1 247.901} C_DIS
LIN {X 0.188,Y -514.972,Z 1032.167,A 0.000,B 0.000,C 90.000,E1 246.102} C_DIS
LIN {X 0.095,Y -513.674,Z 1032.162,A 0.000,B 0.000,C 90.000,E1 245.229} C_DIS
LIN {X -0.143,Y -511.845,Z 1032.156,A 0.000,B 0.000,C 90.000,E1 244.076} C_DIS
LIN {X -0.305,Y -509.459,Z 1032.148,A 0.000,B 0.000,C 90.000,E1 242.615} C_DIS
LIN {X -0.041,Y -506.855,Z 1032.140,A 0.000,B 0.000,C 90.000,E1 241.101} C_DIS
LIN {X -0.076,Y -504.235,Z 1032.131,A 0.000,B 0.000,C 90.000,E1 239.616} C_DIS
LIN {X -0.270,Y -502.619,Z 1032.126,A 0.000,B 0.000,C 90.000,E1 238.742} C_DIS
LIN {X -0.181,Y -500.334,Z 1032.120,A 0.000,B 0.000,C 90.000,E1 237.533} C_DIS
LIN {X -0.146,Y -498.525,Z 1032.115,A 0.000,B 0.000,C 90.000,E1 236.628} C_DIS
LIN {X 0.015,Y -495.406,Z 1032.106,A 0.000,B 0.000,C 90.000,E1 235.102} C_DIS
LIN {X -0.144,Y -492.658,Z 1032.099,A 0.000,B 0.000,C 90.000,E1 233.909} C_DIS
LIN {X 0.021,Y -488.325,Z 1032.089,A 0.000,B 0.000,C 90.000,E1 232.065} C_DIS
LIN {X -0.169,Y -486.184,Z 1032.084,A 0.000,B 0.000,C 90.000,E1 231.170} C_DIS
LIN {X -0.116,Y -481.368,Z 1032.072,A 0.000,B 0.000,C 90.000,E1 229.013} C_DIS
LIN {X -0.033,Y -477.331,Z 1032.062,A 0.000,B 0.000,C 90.000,E1 227.148} C_DIS
LIN {X -0.187,Y -472.148,Z 1032.048,A 0.000,B 0.000,C 90.000,E1 224.676} C_DIS
LIN {X 0.087,Y -470.193,Z 1032.043,A 0.000,B 0.000,C 90.000,E1 223.704} C_DIS
LIN {X -0.152,Y -466.980,Z 1032.034,A 0.000,B 0.000,C 90.000,E1 222.162} C_DIS
LIN {X 0.207,Y -463.716,Z 1032.025,A 0.000,B 0.000,C 90.000,E1 220.539} C_DIS
LIN {X -0.102,Y -460.424,Z 1032.017,A 0.000,B 0.000,C 90.000,E1 218.991} C_DIS
LIN {X -0.205,Y -457.573,Z 1032.010,A 0.000,B 0.000,C 90.000,E1 217.729} C_DIS
LIN {X -0.025,Y -451.328,Z 1031.993,A 0.000,B 0.000,C 90.000,E1 214.818} C_DIS
LIN {X -0.041,Y -447.221,Z 1031.983,A 0.000,B 0.000,C 90.000,E1 212.880} C_DIS
LIN {X -0.083,Y -443.633,Z 1031.974,A 0.000,B 0.000,C 90.000,E1 211.258} C_DIS
LIN {X 0.134,Y -440.803,Z 1031.966,A 0.000,B 0.000,C 90.000,E1 209.922} C_DIS
LIN {X 0.050,Y -438.553,Z 1031.961,A 0.000,B 0.000,C 90.000,E1 208.949} C_DIS
LIN {X -0.031,Y -435.521,Z 1031.954,A 0.000,B 0.000,C 90.000,E1 207.641} C_DIS
LIN {X 0.035,Y -431.792,Z 1031.944,A 0.000,B 0.000,C 90.000,E1 205.976} C_DIS
LIN {X 0.214,Y -427.325,Z 1031.933,A 0.000,B 0.000,C 90.000,E1 203.951} C_DIS
LIN {X -0.052,Y -423.173,Z 1031.922,A 0.000,B 0.000,C 90.000,E1 201.972} C_DIS
LIN {X -0.075,Y -418.060,Z 1031.907,A 0.000,B 0.000,C 90.000,E1 199.268} C_DIS
LIN {X -0.127,Y -413.176,Z 1031.890,A 0.000,B 0.000,C 90.000,E1 196.205} C_DIS
LIN {X 0.201,Y -409.841,Z 1031.875,A 0.000,B 0.000,C 90.000,E1 193.411} C_DIS
LIN {X 0.000,Y -408.635,Z 1031.865,A 0.000,B 0.000,C 90.000,E1 191.715} C_DIS
LIN {X 0.101,Y -408.718,Z 1031.863,A 0.000,B 0.000,C 90.000,E1 191.366} C_DIS
LIN {X 0.173,Y -408.630,Z 1031.860,A 0.000,B 0.000,C 90.000,E1 190.838} C_DIS
LIN {X -0.026,Y -409.044,Z 1031.858,A 0.000,B 0.000,C 90.000,E1 190.423} C_DIS
LIN {X -0.006,Y -409.618,Z 1031.856,A 0.000,B 0.000,C 90.000,E1 190.074} C_DIS
LIN {X -0.041,Y -411.249,Z 1031.853,A 0.000,B 0.000,C 90.000,E1 189.443} C_DIS
LIN {X 0.101,Y -413.486,Z 1031.850,A 0.000,B 0.000,C 90.000,E1 188.916} C_DIS
LIN {X 0.133,Y -416.193,Z 1031.847,A 0.000,B 0.000,C 90.000,E1 188.398} C_DIS
LIN {X -0.172,Y -421.860,Z 1031.842,A 0.000,B 0.000,C 90.000,E1 187.587} C_DIS
LIN {X 0.031,Y -434.400,Z 1031.833,A 0.000,B 0.000,C 90.000,E1 185.910} C_DIS
LIN {X 0.167,Y -447.004,Z 1031.824,A 0.000,B 0.000,C 90.000,E1 184.245} C_DIS
LIN {X 0.106,Y -457.994,Z 1031.816,A 0.000,B 0.000,C 90.000,E1 182.808} C_DIS
LIN {X -0.104,Y -466.344,Z 1031.810,A 0.000,B 0.000,C 90.000,E1 181.718} C_DIS
LIN {X 0.126,Y -473.182,Z 1031.804,A 0.000,B 0.000,C 90.000,E1 180.745} C_DIS
LIN {X 0.106,Y -480.794,Z 1031.798,A 0.000,B 0.000,C 90.000,E1 179.656} C_DIS
LIN {X 0.187,Y -488.083,Z 1031.792,A 0.000,B 0.000,C 90.000,E1 178.568} C_DIS
LIN {X 0.207,Y -494.262,Z 1031.787,A 0.000,B 0.000,C 90.000,E1 177.650} C_DIS
LIN {X -0.195,Y -500.105,Z 1031.782,A 0.000,B 0.000,C 90.000,E1 176.788} C_DIS
LIN {X 0.215,Y -508.236,Z 1031.775,A 0.000,B 0.000,C 90.000,E1 175.412} C_DIS
LIN {X -0.255,Y -512.598,Z 1031.771,A 0.000,B 0.000,C 90.000,E1 174.723} C_DIS
LIN {X -0.092,Y -515.405,Z 1031.768,A 0.000,B 0.000,C 90.000,E1 174.261} C_DIS
LIN {X 0.245,Y -523.863,Z 1031.760,A 0.000,B 0.000,C 90.000,E1 172.761} C_DIS
LIN {X -0.051,Y -531.310,Z 1031.753,A 0.000,B 0.000,C 90.000,E1 171.489} C_DIS
LIN {X -0.149,Y -538.585,Z 1031.746,A 0.000,B 0.000,C 90.000,E1 170.208} C_DIS
LIN {X 0.138,Y -546.613,Z 1031.738,A 0.000,B 0.000,C 90.000,E1 168.757} C_DIS
LIN {X 0.287,Y -552.147,Z 1031.732,A 0.000,B 0.000,C 90.000,E1 167.757} C_DIS
LIN {X -0.157,Y -557.439,Z 1031.727,A 0.000,B 0.000,C 90.000,E1 166.825} C_DIS
LIN {X -0.127,Y -564.009,Z 1031.720,A 0.000,B 0.000,C 90.000,E1 165.574} C_DIS
LIN {X -0.133,Y -570.481,Z 1031.713,A 0.000,B 0.000,C 90.000,E1 164.338} C_DIS
LIN {X 0.112,Y -576.656,Z 1031.706,A 0.000,B 0.000,C 90.000,E1 163.087} C_DIS
LIN {X -0.225,Y -580.541,Z 1031.702,A 0.000,B 0.000,C 90.000,E1 162.308} C_DIS
LIN {X 0.132,Y -584.800,Z 1031.696,A 0.000,B 0.000,C 90.000,E1 161.329} C_DIS
LIN {X 0.291,Y -589.349,Z 1031.690,A 0.000,B 0.000,C 90.000,E1 160.242} C_DIS
LIN {X -0.052,Y -593.707,Z 1031.685,A 0.000,B 0.000,C 90.000,E1 159.209} C_DIS
LIN {X -0.029,Y -596.821,Z 1031.680,A 0.000,B 0.000,C 90.000,E1 158.411} C_DIS
LIN {X 0.024,Y -599.764,Z 1031.676,A 0.000,B 0.000,C 90.000,E1 157.614} C_DIS
LIN {X 0.340,Y -602.544,Z 1031.671,A 0.000,B 0.000,C 90.000,E1 156.794} C_DIS
LIN {X -0.167,Y -605.970,Z 1031.666,A 0.000,B 0.000,C 90.000,E1 155.793} C_DIS
LIN {X 0.176,Y -609.220,Z 1031.660,A 0.000,B 0.000,C 90.000,E1 154.717} C_DIS
LIN {X 0.016,Y -612.234,Z 1031.654,A 0.000,B 0.000,C 90.000,E1 153.691} C_DIS
LIN {X -0.101,Y -615.134,Z 1031.648,A 0.000,B 0.000,C 90.000,E1 152.666} C_DIS
LIN {X -0.221,Y -619.104,Z 1031.640,A 0.000,B 0.000,C 90.000,E1 151.129} C_DIS
LIN {X 0.045,Y -621.066,Z 1031.635,A 0.000,B 0.000,C 90.000,E1 150.333} C_DIS
LIN {X 0.110,Y -624.980,Z 1031.627,A 0.000,B 0.000,C 90.000,E1 148.791} C_DIS
LIN {X -0.268,Y -629.234,Z 1031.617,A 0.000,B 0.000,C 90.000,E1 147.041} C_DIS
LIN {X -0.074,Y -631.663,Z 1031.611,A 0.000,B 0.000,C 90.000,E1 146.008} C_DIS
LIN {X 0.017,Y -635.270,Z 1031.603,A 0.000,B 0.000,C 90.000,E1 144.482} C_DIS
LIN {X 0.037,Y -638.832,Z 1031.594,A 0.000,B 0.000,C 90.000,E1 142.970} C_DIS
LIN {X 0.132,Y -642.378,Z 1031.586,A 0.000,B 0.000,C 90.000,E1 141.457} C_DIS
LIN {X 0.280,Y -645.315,Z 1031.579,A 0.000,B 0.000,C 90.000,E1 140.194} C_DIS
LIN {X -0.020,Y -648.794,Z 1031.571,A 0.000,B 0.000,C 90.000,E1 138.728} C_DIS
LIN {X -0.064,Y -654.818,Z 1031.557,A 0.000,B 0.000,C 90.000,E1 136.257} C_DIS
LIN {X 0.130,Y -660.732,Z 1031.545,A 0.000,B 0.000,C 90.000,E1 134.028} C_DIS
LIN {X 0.060,Y -665.690,Z 1031.535,A 0.000,B 0.000,C 90.000,E1 132.324} C_DIS
LIN {X -0.403,Y -669.297,Z 1031.528,A 0.000,B 0.000,C 90.000,E1 131.148} C_DIS
LIN {X 0.201,Y -672.767,Z 1031.522,A 0.000,B 0.000,C 90.000,E1 129.886} C_DIS
LIN {X -0.067,Y -676.757,Z 1031.514,A 0.000,B 0.000,C 90.000,E1 128.463} C_DIS
LIN {X -0.153,Y -680.569,Z 1031.506,A 0.000,B 0.000,C 90.000,E1 127.030} C_DIS
LIN {X -0.147,Y -684.926,Z 1031.496,A 0.000,B 0.000,C 90.000,E1 125.358} C_DIS
LIN {X -0.134,Y -687.380,Z 1031.491,A 0.000,B 0.000,C 90.000,E1 124.405} C_DIS
LIN {X -0.065,Y -690.379,Z 1031.484,A 0.000,B 0.000,C 90.000,E1 123.214} C_DIS
LIN {X -0.105,Y -693.884,Z 1031.477,A 0.000,B 0.000,C 90.000,E1 121.799} C_DIS
LIN {X 0.020,Y -695.557,Z 1031.473,A 0.000,B 0.000,C 90.000,E1 121.082} C_DIS
LIN {X -0.077,Y -697.048,Z 1031.469,A 0.000,B 0.000,C 90.000,E1 120.384} C_DIS
LIN {X 0.343,Y -698.738,Z 1031.464,A 0.000,B 0.000,C 90.000,E1 119.411} C_DIS
LIN {X -0.168,Y -700.428,Z 1031.457,A 0.000,B 0.000,C 90.000,E1 118.281} C_DIS
LIN {X -0.025,Y -701.410,Z 1031.452,A 0.000,B 0.000,C 90.000,E1 117.334} C_DIS
LIN {X 0.108,Y -702.569,Z 1031.445,A 0.000,B 0.000,C 90.000,E1 116.155} C_DIS
LIN {X -0.083,Y -703.709,Z 1031.438,A 0.000,B 0.000,C 90.000,E1 114.771} C_DIS
LIN {X -0.169,Y -703.561,Z 1031.434,A 0.000,B 0.000,C 90.000,E1 114.079} C_DIS
LIN {X 0.109,Y -702.578,Z 1031.431,A 0.000,B 0.000,C 90.000,E1 113.590} C_DIS
LIN {X -0.257,Y -701.855,Z 1031.430,A 0.000,B 0.000,C 90.000,E1 113.387} C_DIS
LIN {X 0.012,Y -699.186,Z 1031.427,A 0.000,B 0.000,C 90.000,E1 112.898} C_DIS
LIN {X 0.144,Y -698.409,Z 1031.427,A 0.000,B 0.000,C 90.000,E1 112.770} C_DIS
LIN {X 0.275,Y -697.259,Z 1031.426,A 0.000,B 0.000,C 90.000,E1 112.642} C_DIS
LIN {X 0.403,Y -695.521,Z 1031.425,A 0.000,B 0.000,C 90.000,E1 112.514} C_DIS
LIN {X -0.068,Y -690.563,Z 1031.424,A 0.000,B 0.000,C 90.000,E1 112.259} C_DIS
LIN {X 0.138,Y -688.869,Z 1031.423,A 0.000,B 0.000,C 90.000,E1 112.153} C_DIS
LIN {X -0.101,Y -684.370,Z 1031.422,A 0.000,B 0.000,C 90.000,E1 112.025} C_DIS
LIN {X 0.020,Y -675.490,Z 1031.422,A 0.000,B 0.000,C 90.000,E1 111.897} C_DIS
LIN {X -0.029,Y -612.319,Z 1031.422,A 0.000,B 0.000,C 90.000,E1 111.897} C_DIS
LIN {X -0.305,Y -609.699,Z 1031.421,A 0.000,B 0.000,C 90.000,E1 111.844} C_DIS
LIN {X -0.051,Y -604.555,Z 1031.420,A 0.000,B 0.000,C 90.000,E1 111.642} C_DIS
LIN {X -0.238,Y -598.228,Z 1031.419,A 0.000,B 0.000,C 90.000,E1 111.354} C_DIS
LIN {X 0.064,Y -592.618,Z 1031.417,A 0.000,B 0.000,C 90.000,E1 110.972} C_DIS
LIN {X -0.171,Y -585.357,Z 1031.413,A 0.000,B 0.000,C 90.000,E1 110.429} C_DIS
LIN {X -0.120,Y -577.541,Z 1031.410,A 0.000,B 0.000,C 90.000,E1 109.758} C_DIS
LIN {X -0.241,Y -570.152,Z 1031.407,A 0.000,B 0.000,C 90.000,E1 109.214} C_DIS
LIN {X -0.156,Y -561.815,Z 1031.404,A 0.000,B 0.000,C 90.000,E1 108.725} C_DIS
LIN {X -0.017,Y -555.019,Z 1031.402,A 0.000,B 0.000,C 90.000,E1 108.362} C_DIS
LIN {X -0.030,Y -550.058,Z 1031.400,A 0.000,B 0.000,C 90.000,E1 108.055} C_DIS
LIN {X 0.128,Y -549.107,Z 1031.400,A 0.000,B 0.000,C 90.000,E1 107.946} C_DIS
LIN {X 0.207,Y -548.138,Z 1031.399,A 0.000,B 0.000,C 90.000,E1 107.819} C_DIS
LIN {X 0.164,Y -548.123,Z 1031.399,A 0.000,B 0.000,C 90.000,E1 107.819} C_DIS
LIN {X 0.251,Y -547.752,Z 1031.397,A 0.000,B 0.000,C 90.000,E1 107.511} C_DIS
LIN {X 0.109,Y -548.767,Z 1031.384,A 0.000,B 0.000,C 90.000,E1 105.134} C_DIS
LIN {X 0.147,Y -550.146,Z 1031.372,A 0.000,B 0.000,C 90.000,E1 102.883} C_DIS
LIN {X 0.204,Y -552.618,Z 1031.356,A 0.000,B 0.000,C 90.000,E1 100.074} C_DIS
LIN {X 0.079,Y -554.175,Z 1031.348,A 0.000,B 0.000,C 90.000,E1 98.690} C_DIS
LIN {X 0.127,Y -556.069,Z 1031.339,A 0.000,B 0.000,C 90.000,E1 97.011} C_DIS
